# B&R Automation Studio project 8238 (part 18)

#### mnParam_GetCsvDat.st - Parsen einer CSV-Zeile
```iecst
(********************************************************************
 * COPYRIGHT -- Microsoft
 ********************************************************************
 * Library: mnParamLib
 * File: mnParam_GetCsvDat.st
 * Author: hunholz
 * Created: July 25, 2011
 * Changed: Mar 29, 2012
 ********************************************************************
 * Implementation of library mnParamLib
 ********************************************************************)

(* Parsen einer CSV-Zeile *)
FUNCTION_BLOCK mnParam_GetCsvDat

	IF enable THEN

		status := ERR_OK;

		RowType := 0;

		brsmemset(ADR(HeaderVersion), 0, SIZEOF(HeaderVersion));
		brsmemset(ADR(HeaderMachineNo), 0, SIZEOF(HeaderMachineNo));
		brsmemset(ADR(HeaderTime), 0, SIZEOF(HeaderTime));
		brsmemset(ADR(ContainerRow), 0, SIZEOF(ContainerRow));
		brsmemset(ADR(LogicalStructRow), 0, SIZEOF(LogicalStructRow));
		brsmemset(ADR(ParamNumRow), 0, SIZEOF(ParamNumRow));
		brsmemset(ADR(ParamStringRow), 0, SIZEOF(ParamStringRow));
		brsmemset(ADR(CsvNumRow), 0, SIZEOF(CsvNumRow));
		brsmemset(ADR(CsvStringRow), 0, SIZEOF(CsvStringRow));
		brsmemset(ADR(CsvIPRow),0,SIZEOF(CsvIPRow));
		brsmemset(ADR(csvTextRow),0,SIZEOF(csvTextRow));
		brsmemset(ADR(csvHelpTextRow), 0, SIZEOF(csvHelpTextRow));
		brsmemset(ADR(CsvCProw), 0, SIZEOF(CsvCProw));

		_pUtfCsvString := ADR(utfCsvString);

		_GetNextSubstring.enable := TRUE;
		_GetNextSubstring(pUtfCsvString := _pUtfCsvString);

		_utfRowType := "";

		brwcsncpy(ADR(_utfRowType), _GetNextSubstring.pUtfCsvSubstring, MIN(_GetNextSubstring.Length, 15));
		brwcsconv(ADR(_sRowType), ADR(_utfRowType), 1);

		_diRowType := atoi(ADR(_sRowType) );

		IF _diRowType = MNPARAM_CSV_FILEEND THEN

			// FileEnde
			RowType := MNPARAM_CSV_FILEEND;
			// Keine Rückgabewerte

		ELSIF _diRowType = MNPARAM_CSV_COMMENT THEN

			// Kommentarzeile
			RowType := MNPARAM_CSV_COMMENT;

		ELSIF _diRowType = MNPARAM_CSV_HEADER_VERSION THEN

			// Version Datenmodell
			RowType := MNPARAM_CSV_HEADER_VERSION;

			IF NOT _GetNextSubstring.EndOfLine THEN

				_GetNextSubstring(pUtfCsvString := _pUtfCsvString);

				_utfSubString := "";

				brwcsncpy(ADR(_utfSubString), _GetNextSubstring.pUtfCsvSubstring, MIN(_GetNextSubstring.Length, 63));
				brwcsconv(ADR(_sSubString), ADR(_utfSubString), 1);
				_diVersion := atoi(ADR(_sSubString) );

				HeaderVersion.wVersion := DINT_TO_UINT(LIMIT(0, _diVersion, 65535));

			END_IF

			IF NOT _GetNextSubstring.EndOfLine THEN

				_GetNextSubstring(pUtfCsvString := _pUtfCsvString);

				_utfSubString := "";

				brwcsncpy(ADR(_utfSubString), _GetNextSubstring.pUtfCsvSubstring, MIN(_GetNextSubstring.Length, 63));
				brwcsconv(ADR(_sSubString), ADR(_utfSubString), 1);

				_atodt(pStr := ADR(_sSubString));
				HeaderVersion.dtTimestamp := _atodt.dtTimeStamp;

			END_IF

			IF NOT _GetNextSubstring.EndOfLine THEN

				_GetNextSubstring(pUtfCsvString := _pUtfCsvString);

				brwcsncpy(ADR(HeaderVersion.utfMachineType), _GetNextSubstring.pUtfCsvSubstring, MIN(_GetNextSubstring.Length,11));

			END_IF

			IF NOT _GetNextSubstring.EndOfLine THEN

				_GetNextSubstring(pUtfCsvString := _pUtfCsvString);

				brwcsncpy(ADR(HeaderVersion.utfMachineSubType), _GetNextSubstring.pUtfCsvSubstring, MIN(_GetNextSubstring.Length,11));

			END_IF

		ELSIF _diRowType = MNPARAM_CSV_HEADER_MACHINENO THEN

			// Maschinennummer
			RowType := MNPARAM_CSV_HEADER_MACHINENO;

			IF NOT _GetNextSubstring.EndOfLine THEN

				_GetNextSubstring(pUtfCsvString := _pUtfCsvString);

				brwcsncpy(ADR(HeaderMachineNo.utfMachineNo), _GetNextSubstring.pUtfCsvSubstring, MIN(_GetNextSubstring.Length,15));

			END_IF

		ELSIF _diRowType = MNPARAM_CSV_HEADER_TIMESTAMP THEN

			// TimeStamp
			RowType := MNPARAM_CSV_HEADER_TIMESTAMP;

			IF NOT _GetNextSubstring.EndOfLine THEN

				_GetNextSubstring(pUtfCsvString := _pUtfCsvString);

				_utfSubString := "";

				brwcsncpy(ADR(_utfSubString), _GetNextSubstring.pUtfCsvSubstring, MIN(_GetNextSubstring.Length, 63));
				brwcsconv(ADR(_sSubString), ADR(_utfSubString), 1);

				_atodt(pStr := ADR(_sSubString));
				HeaderTime.dtTimestamp := _atodt.dtTimeStamp;

			END_IF

		ELSIF _diRowType = MNPARAM_CSV_LANGUAGEDEF THEN

			// Sprachdefinition
			RowType := MNPARAM_CSV_LANGUAGEDEF;

			IF NOT _GetNextSubstring.EndOfLine THEN

				_GetNextSubstring(pUtfCsvString := _pUtfCsvString);

				_utfSubString := "";

				brwcsncpy(ADR(_utfSubString), _GetNextSubstring.pUtfCsvSubstring, MIN(_GetNextSubstring.Length, 63));
				brwcsconv(ADR(_sSubString), ADR(_utfSubString), 1);
				_diNum := atoi(ADR(_sSubString) );

				CsvLCIDrow.LCID := DINT_TO_UINT(LIMIT(0, _diNum, 65535));

			END_IF

			IF NOT _GetNextSubstring.EndOfLine THEN

				_GetNextSubstring(pUtfCsvString := _pUtfCsvString);

				brwcsncpy(ADR(CsvLCIDrow.utfName), _GetNextSubstring.pUtfCsvSubstring, MIN(_GetNextSubstring.Length, 31));

			END_IF

		ELSIF _diRowType = MNPARAM_CSV_LAN_HELPTEXT THEN

			// Sprachhilfstext
			RowType := MNPARAM_CSV_LAN_HELPTEXT;

			IF NOT _GetNextSubstring.EndOfLine THEN

				_GetNextSubstring(pUtfCsvString := _pUtfCsvString);

				_utfSubString := "";

				brwcsncpy(ADR(_utfSubString), _GetNextSubstring.pUtfCsvSubstring, MIN(_GetNextSubstring.Length, 63));
				brwcsconv(ADR(_sSubString), ADR(_utfSubString), 1);
				_diNum := atoi(ADR(_sSubString) );

				csvHelpTextRow.LCID := DINT_TO_UINT(LIMIT(0, _diNum, 65535));

			END_IF

			IF NOT _GetNextSubstring.EndOfLine THEN

				_GetNextSubstring(pUtfCsvString := _pUtfCsvString);

				_utfSubString := "";

				brwcsncpy(ADR(_utfSubString), _GetNextSubstring.pUtfCsvSubstring, MIN(_GetNextSubstring.Length, 63));
				brwcsconv(ADR(_sSubString), ADR(_utfSubString), 1);
				_diNum := atoi(ADR(_sSubString) );

				csvHelpTextRow.FunctionID := DINT_TO_UINT(LIMIT(0, _diNum, 65535));

			END_IF

			IF NOT _GetNextSubstring.EndOfLine THEN

				_GetNextSubstring(pUtfCsvString := _pUtfCsvString);

				_utfSubString := "";

				brwcsncpy(ADR(_utfSubString), _GetNextSubstring.pUtfCsvSubstring, MIN(_GetNextSubstring.Length, 63));
				brwcsconv(ADR(_sSubString), ADR(_utfSubString), 1);
				_diNum := atoi(ADR(_sSubString) );

				csvHelpTextRow.TextNo := DINT_TO_UINT(LIMIT(0, _diNum, 65535));

			END_IF

			IF NOT _GetNextSubstring.EndOfLine THEN

				_GetNextSubstring(pUtfCsvString := _pUtfCsvString);

				brwcsncpy(ADR(csvHelpTextRow.utfHelpText), _GetNextSubstring.pUtfCsvSubstring, MIN(_GetNextSubstring.Length, 255));

			END_IF

		ELSIF _diRowType = MNPARAM_CSV_LAN_TEXT THEN

			// Sprachtext
			RowType := MNPARAM_CSV_LAN_TEXT;

			IF NOT _GetNextSubstring.EndOfLine THEN

				_GetNextSubstring(pUtfCsvString := _pUtfCsvString);

				_utfSubString := "";

				brwcsncpy(ADR(_utfSubString), _GetNextSubstring.pUtfCsvSubstring, MIN(_GetNextSubstring.Length, 63));
				brwcsconv(ADR(_sSubString), ADR(_utfSubString), 1);
				_diNum := atoi(ADR(_sSubString) );

				csvTextRow.LCID := DINT_TO_UINT(LIMIT(0, _diNum, 65535));

			END_IF

			IF NOT _GetNextSubstring.EndOfLine THEN

				_GetNextSubstring(pUtfCsvString := _pUtfCsvString);

				_utfSubString := "";

				brwcsncpy(ADR(_utfSubString), _GetNextSubstring.pUtfCsvSubstring, MIN(_GetNextSubstring.Length, 63));
				brwcsconv(ADR(_sSubString), ADR(_utfSubString), 1);
				_diNum := atoi(ADR(_sSubString) );

				csvTextRow.FunctionID := DINT_TO_UINT(LIMIT(0, _diNum, 65535));

			END_IF

			IF NOT _GetNextSubstring.EndOfLine THEN

				_GetNextSubstring(pUtfCsvString := _pUtfCsvString);

				_utfSubString := "";

				brwcsncpy(ADR(_utfSubString), _GetNextSubstring.pUtfCsvSubstring, MIN(_GetNextSubstring.Length, 63));
				brwcsconv(ADR(_sSubString), ADR(_utfSubString), 1);
				_diNum := atoi(ADR(_sSubString) );

				csvTextRow.TextNo := DINT_TO_UINT(LIMIT(0, _diNum, 65535));

			END_IF

			IF NOT _GetNextSubstring.EndOfLine THEN

				_GetNextSubstring(pUtfCsvString := _pUtfCsvString);

				brwcsncpy(ADR(csvTextRow.utfText), _GetNextSubstring.pUtfCsvSubstring, MIN(_GetNextSubstring.Length, 63));

			END_IF

		ELSIF _diRowType = MNPARAM_CSV_DEF_CONTAINER THEN

			// Containerbeschreibung
			RowType := MNPARAM_CSV_DEF_CONTAINER;

			// Container ID
			IF NOT _GetNextSubstring.EndOfLine THEN

				_GetNextSubstring(pUtfCsvString := _pUtfCsvString);

				_utfSubString := "";

				brwcsncpy(ADR(_utfSubString), _GetNextSubstring.pUtfCsvSubstring, MIN(_GetNextSubstring.Length, 63));
				brwcsconv(ADR(_sSubString), ADR(_utfSubString), 1);
				_diNum := atoi(ADR(_sSubString) );

				ContainerRow.siContainerID := DINT_TO_SINT(LIMIT(-128, _diNum, 127));

			END_IF

			// DirectParam
			IF NOT _GetNextSubstring.EndOfLine THEN

				_GetNextSubstring(pUtfCsvString := _pUtfCsvString);

				_utfSubString := "";

				brwcsncpy(ADR(_utfSubString), _GetNextSubstring.pUtfCsvSubstring, MIN(_GetNextSubstring.Length, 63));
				brwcsconv(ADR(_sSubString), ADR(_utfSubString), 1);
				_diNum := atoi(ADR(_sSubString) );

				ContainerRow.bDirectParam := DINT_TO_BOOL(LIMIT(0, _diNum, 1));

			END_IF

			// Name Data Obj
			IF NOT _GetNextSubstring.EndOfLine THEN

				_GetNextSubstring(pUtfCsvString := _pUtfCsvString);

				_utfSubString := "";

				brwcsncpy(ADR(_utfDataObj), _GetNextSubstring.pUtfCsvSubstring, MIN(_GetNextSubstring.Length, 11));
				brwcsconv(ADR(ContainerRow.sNameDataObj), ADR(_utfDataObj), 1);

			END_IF

			// Name Csv File
			IF NOT _GetNextSubstring.EndOfLine THEN

				_GetNextSubstring(pUtfCsvString := _pUtfCsvString);

				_utfSubString := "";

				brwcsncpy(ADR(_utfSubString), _GetNextSubstring.pUtfCsvSubstring, MIN(_GetNextSubstring.Length, 31));
				brwcsconv(ADR(ContainerRow.sNameCsv), ADR(_utfSubString), 1);

			END_IF

			// Min Bound
			IF NOT _GetNextSubstring.EndOfLine THEN

				_GetNextSubstring(pUtfCsvString := _pUtfCsvString);

				_utfSubString := "";

				brwcsncpy(ADR(_utfSubString), _GetNextSubstring.pUtfCsvSubstring, MIN(_GetNextSubstring.Length, 63));
				brwcsconv(ADR(_sSubString), ADR(_utfSubString), 1);
				_diNum := atoi(ADR(_sSubString) );

				ContainerRow.wMinBound := DINT_TO_UINT(LIMIT(0, _diNum, 65535));

			END_IF

			// Dimension
			IF NOT _GetNextSubstring.EndOfLine THEN

				_GetNextSubstring(pUtfCsvString := _pUtfCsvString);

				_utfSubString := "";

				brwcsncpy(ADR(_utfSubString), _GetNextSubstring.pUtfCsvSubstring, MIN(_GetNextSubstring.Length, 63));
				brwcsconv(ADR(_sSubString), ADR(_utfSubString), 1);
				_diNum := atoi(ADR(_sSubString) );

				ContainerRow.wDimension := DINT_TO_UINT(LIMIT(0, _diNum, 65535));

			END_IF

			// Struct Root
			IF NOT _GetNextSubstring.EndOfLine THEN

				_GetNextSubstring(pUtfCsvString := _pUtfCsvString);

				_utfSubString := "";

				brwcsncpy(ADR(_utfSubString), _GetNextSubstring.pUtfCsvSubstring, MIN(_GetNextSubstring.Length, 31));
				brwcsconv(ADR(ContainerRow.sStrucRoot), ADR(_utfSubString), 1);

			END_IF

			IF NOT _GetNextSubstring.EndOfLine THEN
				_GetNextSubstring(pUtfCsvString := _pUtfCsvString);
			END_IF

			// Anzahl der Numparameter
			IF NOT _GetNextSubstring.EndOfLine THEN

				_GetNextSubstring(pUtfCsvString := _pUtfCsvString);

				_utfSubString := "";

				brwcsncpy(ADR(_utfSubString), _GetNextSubstring.pUtfCsvSubstring, MIN(_GetNextSubstring.Length, 63));
				brwcsconv(ADR(_sSubString), ADR(_utfSubString), 1);

				ContainerRow.lCountNum := atoi(ADR(_sSubString) );

			END_IF

			// Anzahl der Stringparameter
			IF NOT _GetNextSubstring.EndOfLine THEN

				_GetNextSubstring(pUtfCsvString := _pUtfCsvString);

				_utfSubString := "";

				brwcsncpy(ADR(_utfSubString), _GetNextSubstring.pUtfCsvSubstring, MIN(_GetNextSubstring.Length, 63));
				brwcsconv(ADR(_sSubString), ADR(_utfSubString), 1);

				ContainerRow.lCountString := atoi(ADR(_sSubString) );

			END_IF

		ELSIF _diRowType = MNPARAM_CSV_DEF_LOGSTRUC THEN

			// Logische Struktur
			RowType := MNPARAM_CSV_DEF_LOGSTRUC;

			// Index
			IF NOT _GetNextSubstring.EndOfLine THEN

				_GetNextSubstring(pUtfCsvString := _pUtfCsvString);

				_utfSubString := "";

				brwcsncpy(ADR(_utfSubString), _GetNextSubstring.pUtfCsvSubstring, MIN(_GetNextSubstring.Length, 63));
				brwcsconv(ADR(_sSubString), ADR(_utfSubString), 1);
				_diNum := atoi(ADR(_sSubString) );

				LogicalStructRow.wLogStrucNo := DINT_TO_UINT(LIMIT(0, _diNum, 65535));

			END_IF

			// Min Bound
			IF NOT _GetNextSubstring.EndOfLine THEN

				_GetNextSubstring(pUtfCsvString := _pUtfCsvString);

				_utfSubString := "";

				brwcsncpy(ADR(_utfSubString), _GetNextSubstring.pUtfCsvSubstring, MIN(_GetNextSubstring.Length, 63));
				brwcsconv(ADR(_sSubString), ADR(_utfSubString), 1);
				_diNum := atoi(ADR(_sSubString) );

				LogicalStructRow.wMinBound := DINT_TO_UINT(LIMIT(0, _diNum, 65535));

			END_IF

			// Dimension
			IF NOT _GetNextSubstring.EndOfLine THEN

				_GetNextSubstring(pUtfCsvString := _pUtfCsvString);

				_utfSubString := "";

				brwcsncpy(ADR(_utfSubString), _GetNextSubstring.pUtfCsvSubstring, MIN(_GetNextSubstring.Length, 63));
				brwcsconv(ADR(_sSubString), ADR(_utfSubString), 1);
				_diNum := atoi(ADR(_sSubString) );

				LogicalStructRow.wDimension := DINT_TO_UINT(LIMIT(0, _diNum, 65535));

			END_IF

			// Referenz
			IF NOT _GetNextSubstring.EndOfLine THEN

				_GetNextSubstring(pUtfCsvString := _pUtfCsvString);

				_utfSubString := "";

				brwcsncpy(ADR(_utfSubString), _GetNextSubstring.pUtfCsvSubstring, MIN(_GetNextSubstring.Length, 63));
				brwcsconv(ADR(_sSubString), ADR(_utfSubString), 1);
				_diNum := atoi(ADR(_sSubString) );

				LogicalStructRow.iReferenz := DINT_TO_INT(LIMIT(-32768, _diNum, 32767));

			END_IF

			// Ref Visible
			IF NOT _GetNextSubstring.EndOfLine THEN

				_GetNextSubstring(pUtfCsvString := _pUtfCsvString);

				_utfSubString := "";

				brwcsncpy(ADR(_utfSubString), _GetNextSubstring.pUtfCsvSubstring, MIN(_GetNextSubstring.Length, 63));
				brwcsconv(ADR(_sSubString), ADR(_utfSubString), 1);
				_diNum := atoi(ADR(_sSubString) );

				LogicalStructRow.wRefVisible := DINT_TO_UINT(LIMIT(0, _diNum, 65535));

			END_IF

			// Ref Text
			IF NOT _GetNextSubstring.EndOfLine THEN

				_GetNextSubstring(pUtfCsvString := _pUtfCsvString);

				_utfSubString := "";

				brwcsncpy(ADR(_utfSubString), _GetNextSubstring.pUtfCsvSubstring, MIN(_GetNextSubstring.Length, 63));
				brwcsconv(ADR(_sSubString), ADR(_utfSubString), 1);
				_diNum := atoi(ADR(_sSubString) );

				LogicalStructRow.wRefText := DINT_TO_UINT(LIMIT(0, _diNum, 65535));

			END_IF

			// WriteAccess
			IF NOT _GetNextSubstring.EndOfLine THEN

				_GetNextSubstring(pUtfCsvString := _pUtfCsvString);

				_utfSubString := "";

				brwcsncpy(ADR(_utfSubString), _GetNextSubstring.pUtfCsvSubstring, MIN(_GetNextSubstring.Length, 63));
				brwcsconv(ADR(_sSubString), ADR(_utfSubString), 1);
				_diNum := atoi(ADR(_sSubString) );

				LogicalStructRow.siWriteAccess := DINT_TO_SINT(LIMIT(-128, _diNum, 127));

			END_IF

			// VisibleAccess
			IF NOT _GetNextSubstring.EndOfLine THEN

				_GetNextSubstring(pUtfCsvString := _pUtfCsvString);

				_utfSubString := "";

				brwcsncpy(ADR(_utfSubString), _GetNextSubstring.pUtfCsvSubstring, MIN(_GetNextSubstring.Length, 63));
				brwcsconv(ADR(_sSubString), ADR(_utfSubString), 1);
				_diNum := atoi(ADR(_sSubString) );

				LogicalStructRow.siVisibleAccess := DINT_TO_SINT(LIMIT(-128, _diNum, 127));

			END_IF

			// Format Array
			IF NOT _GetNextSubstring.EndOfLine THEN

				_GetNextSubstring(pUtfCsvString := _pUtfCsvString);

				_utfSubString := "";

				brwcsncpy(ADR(_utfSubString), _GetNextSubstring.pUtfCsvSubstring, MIN(_GetNextSubstring.Length, 63));
				brwcsconv(ADR(_sSubString), ADR(_utfSubString), 1);
				_diNum := atoi(ADR(_sSubString) );

				LogicalStructRow.bFormatArray := DINT_TO_USINT(LIMIT(0, _diNum, 255));

			END_IF

			// Machine Sub Type
			IF NOT _GetNextSubstring.EndOfLine THEN

				_GetNextSubstring(pUtfCsvString := _pUtfCsvString);

				brwcsncpy(ADR(LogicalStructRow.utfMachineSubType), _GetNextSubstring.pUtfCsvSubstring, MIN(_GetNextSubstring.Length, 11));

			END_IF

			// LogStructName
			IF NOT _GetNextSubstring.EndOfLine THEN

				_GetNextSubstring(pUtfCsvString := _pUtfCsvString);

				brwcsncpy(ADR(LogicalStructRow.utfLogStrucName), _GetNextSubstring.pUtfCsvSubstring, MIN(_GetNextSubstring.Length, 31));

			END_IF

		ELSIF _diRowType = MNPARAM_CSV_DEF_STRING THEN

			// String
			RowType := MNPARAM_CSV_DEF_STRING;

			// Index
			IF NOT _GetNextSubstring.EndOfLine THEN

				_GetNextSubstring(pUtfCsvString := _pUtfCsvString);

				_utfSubString := "";

				brwcsncpy(ADR(_utfSubString), _GetNextSubstring.pUtfCsvSubstring, MIN(_GetNextSubstring.Length, 63));
				brwcsconv(ADR(_sSubString), ADR(_utfSubString), 1);
				_diNum := atoi(ADR(_sSubString) );

				ParamStringRow.wIdxStringPar := DINT_TO_UINT(LIMIT(0, _diNum, 65535));

			END_IF

			// Function ID
			IF NOT _GetNextSubstring.EndOfLine THEN

				_GetNextSubstring(pUtfCsvString := _pUtfCsvString);

				_utfSubString := "";

				brwcsncpy(ADR(_utfSubString), _GetNextSubstring.pUtfCsvSubstring, MIN(_GetNextSubstring.Length, 63));
				brwcsconv(ADR(_sSubString), ADR(_utfSubString), 1);
				_diNum := atoi(ADR(_sSubString) );

				ParamStringRow.wFunction_ID := DINT_TO_UINT(LIMIT(0, _diNum, 65535));

			END_IF

			// Parameter No
			IF NOT _GetNextSubstring.EndOfLine THEN

				_GetNextSubstring(pUtfCsvString := _pUtfCsvString);

				_utfSubString := "";

				brwcsncpy(ADR(_utfSubString), _GetNextSubstring.pUtfCsvSubstring, MIN(_GetNextSubstring.Length, 63));
				brwcsconv(ADR(_sSubString), ADR(_utfSubString), 1);
				_diNum := atoi(ADR(_sSubString) );

				ParamStringRow.wParNo := DINT_TO_UINT(LIMIT(0, _diNum, 65535));

			END_IF

			// Länge
			IF NOT _GetNextSubstring.EndOfLine THEN

				_GetNextSubstring(pUtfCsvString := _pUtfCsvString);

				_utfSubString := "";

				brwcsncpy(ADR(_utfSubString), _GetNextSubstring.pUtfCsvSubstring, MIN(_GetNextSubstring.Length, 63));
				brwcsconv(ADR(_sSubString), ADR(_utfSubString), 1);
				_diNum := atoi(ADR(_sSubString) );

				ParamStringRow.bLenght := DINT_TO_USINT(LIMIT(0, _diNum, 255));

			END_IF

			// WriteAccess
			IF NOT _GetNextSubstring.EndOfLine THEN

				_GetNextSubstring(pUtfCsvString := _pUtfCsvString);

				_utfSubString := "";

				brwcsncpy(ADR(_utfSubString), _GetNextSubstring.pUtfCsvSubstring, MIN(_GetNextSubstring.Length, 63));
				brwcsconv(ADR(_sSubString), ADR(_utfSubString), 1);
				_diNum := atoi(ADR(_sSubString) );

				ParamStringRow.siWriteAccess := DINT_TO_SINT(LIMIT(-128, _diNum, 127));

			END_IF

			// VisibleAccess
			IF NOT _GetNextSubstring.EndOfLine THEN

				_GetNextSubstring(pUtfCsvString := _pUtfCsvString);

				_utfSubString := "";

				brwcsncpy(ADR(_utfSubString), _GetNextSubstring.pUtfCsvSubstring, MIN(_GetNextSubstring.Length, 63));
				brwcsconv(ADR(_sSubString), ADR(_utfSubString), 1);
				_diNum := atoi(ADR(_sSubString) );

				ParamStringRow.siVisibleAccess := DINT_TO_SINT(LIMIT(-128, _diNum, 127));

			END_IF

			// Adresse
			IF NOT _GetNextSubstring.EndOfLine THEN

				_GetNextSubstring(pUtfCsvString := _pUtfCsvString);

				_utfSubString := "";

				brwcsncpy(ADR(_utfSubString), _GetNextSubstring.pUtfCsvSubstring, MIN(_GetNextSubstring.Length, 63));
				brwcsconv(ADR(ParamStringRow.sAdresse), ADR(_utfSubString), 1);

			END_IF

			// Min Bound
			IF NOT _GetNextSubstring.EndOfLine THEN

				_GetNextSubstring(pUtfCsvString := _pUtfCsvString);

				_utfSubString := "";

				brwcsncpy(ADR(_utfSubString), _GetNextSubstring.pUtfCsvSubstring, MIN(_GetNextSubstring.Length, 63));
				brwcsconv(ADR(_sSubString), ADR(_utfSubString), 1);
				_diNum := atoi(ADR(_sSubString) );

				ParamStringRow.wMinBound := DINT_TO_UINT(LIMIT(0, _diNum, 65535));

			END_IF

			// Dimension
			IF NOT _GetNextSubstring.EndOfLine THEN

				_GetNextSubstring(pUtfCsvString := _pUtfCsvString);

				_utfSubString := "";

				brwcsncpy(ADR(_utfSubString), _GetNextSubstring.pUtfCsvSubstring, MIN(_GetNextSubstring.Length, 63));
				brwcsconv(ADR(_sSubString), ADR(_utfSubString), 1);
				_diNum := atoi(ADR(_sSubString) );

				ParamStringRow.wDimension := DINT_TO_UINT(LIMIT(0, _diNum, 65535));

			END_IF

			// Referenz
			IF NOT _GetNextSubstring.EndOfLine THEN

				_GetNextSubstring(pUtfCsvString := _pUtfCsvString);

				_utfSubString := "";

				brwcsncpy(ADR(_utfSubString), _GetNextSubstring.pUtfCsvSubstring, MIN(_GetNextSubstring.Length, 63));
				brwcsconv(ADR(_sSubString), ADR(_utfSubString), 1);
				_diNum := atoi(ADR(_sSubString) );

				ParamStringRow.wReferenz := DINT_TO_UINT(LIMIT(0, _diNum, 65535));

			END_IF

			// Def. Value
			IF NOT _GetNextSubstring.EndOfLine THEN

				_GetNextSubstring(pUtfCsvString := _pUtfCsvString);

				brwcsncpy(ADR(ParamStringRow.utfDefValue), _GetNextSubstring.pUtfCsvSubstring, MIN(_GetNextSubstring.Length, 31));

			END_IF

			// Machine Sub Type
			IF NOT _GetNextSubstring.EndOfLine THEN

				_GetNextSubstring(pUtfCsvString := _pUtfCsvString);

				brwcsncpy(ADR(ParamStringRow.utfMachineSubType), _GetNextSubstring.pUtfCsvSubstring, MIN(_GetNextSubstring.Length, 11));

			END_IF

			// RefVisible
			IF NOT _GetNextSubstring.EndOfLine THEN

				_GetNextSubstring(pUtfCsvString := _pUtfCsvString);

				_utfSubString := "";

				brwcsncpy(ADR(_utfSubString), _GetNextSubstring.pUtfCsvSubstring, MIN(_GetNextSubstring.Length, 63));
				brwcsconv(ADR(_sSubString), ADR(_utfSubString), 1);
				_diNum := atoi(ADR(_sSubString) );

				ParamStringRow.wRefVisible := DINT_TO_UINT(LIMIT(0, _diNum, 65535));

			END_IF

			// RefVisible
			IF NOT _GetNextSubstring.EndOfLine THEN

				_GetNextSubstring(pUtfCsvString := _pUtfCsvString);

				_utfSubString := "";

				brwcsncpy(ADR(_utfSubString), _GetNextSubstring.pUtfCsvSubstring, MIN(_GetNextSubstring.Length, 63));
				brwcsconv(ADR(_sSubString), ADR(_utfSubString), 1);
				_diNum := atoi(ADR(_sSubString) );

				ParamStringRow.wRefVisibleType := DINT_TO_UINT(LIMIT(0, _diNum, 65535));

			END_IF

			// RefText
			IF NOT _GetNextSubstring.EndOfLine THEN

				_GetNextSubstring(pUtfCsvString := _pUtfCsvString);

				_utfSubString := "";

				brwcsncpy(ADR(_utfSubString), _GetNextSubstring.pUtfCsvSubstring, MIN(_GetNextSubstring.Length, 63));
				brwcsconv(ADR(_sSubString), ADR(_utfSubString), 1);
				_diNum := atoi(ADR(_sSubString) );

				ParamStringRow.wRefText := DINT_TO_UINT(LIMIT(0, _diNum, 65535));

			END_IF

		ELSIF _diRowType = MNPARAM_CSV_DEF_NUM OR _diRowType = MNPARAM_CSV_DEF_REAL THEN

			// Logische Struktur
			RowType := DINT_TO_UINT(_diRowType);
			ParamNumRow.bRowType := UINT_TO_USINT(RowType - MNPARAM_CSV_DEF_NUM);

			// Index
			IF NOT _GetNextSubstring.EndOfLine THEN

				_GetNextSubstring(pUtfCsvString := _pUtfCsvString);

				_utfSubString := "";

				brwcsncpy(ADR(_utfSubString), _GetNextSubstring.pUtfCsvSubstring, MIN(_GetNextSubstring.Length, 63));
				brwcsconv(ADR(_sSubString), ADR(_utfSubString), 1);
				_diNum := atoi(ADR(_sSubString) );

				ParamNumRow.wIdxNumPar := DINT_TO_UINT(LIMIT(0, _diNum, 65535));

			END_IF

			// Function ID
			IF NOT _GetNextSubstring.EndOfLine THEN

				_GetNextSubstring(pUtfCsvString := _pUtfCsvString);

				_utfSubString := "";

				brwcsncpy(ADR(_utfSubString), _GetNextSubstring.pUtfCsvSubstring, MIN(_GetNextSubstring.Length, 63));
				brwcsconv(ADR(_sSubString), ADR(_utfSubString), 1);
				_diNum := atoi(ADR(_sSubString) );

				ParamNumRow.wFunction_ID := DINT_TO_UINT(LIMIT(0, _diNum, 65535));

			END_IF

			// Parameter No
			IF NOT _GetNextSubstring.EndOfLine THEN

				_GetNextSubstring(pUtfCsvString := _pUtfCsvString);

				_utfSubString := "";

				brwcsncpy(ADR(_utfSubString), _GetNextSubstring.pUtfCsvSubstring, MIN(_GetNextSubstring.Length, 63));
				brwcsconv(ADR(_sSubString), ADR(_utfSubString), 1);
				_diNum := atoi(ADR(_sSubString) );

				ParamNumRow.wParNo := DINT_TO_UINT(LIMIT(0, _diNum, 65535));

			END_IF

			// WriteAccess
			IF NOT _GetNextSubstring.EndOfLine THEN

				_GetNextSubstring(pUtfCsvString := _pUtfCsvString);

				_utfSubString := "";

				brwcsncpy(ADR(_utfSubString), _GetNextSubstring.pUtfCsvSubstring, MIN(_GetNextSubstring.Length, 63));
				brwcsconv(ADR(_sSubString), ADR(_utfSubString), 1);
				_diNum := atoi(ADR(_sSubString) );

				ParamNumRow.siWriteAccess := DINT_TO_SINT(LIMIT(-128, _diNum, 127));

			END_IF

			// VisibleAccess
			IF NOT _GetNextSubstring.EndOfLine THEN

				_GetNextSubstring(pUtfCsvString := _pUtfCsvString);

				_utfSubString := "";

				brwcsncpy(ADR(_utfSubString), _GetNextSubstring.pUtfCsvSubstring, MIN(_GetNextSubstring.Length, 63));
				brwcsconv(ADR(_sSubString), ADR(_utfSubString), 1);
				_diNum := atoi(ADR(_sSubString) );

				ParamNumRow.siVisibleAccess := DINT_TO_SINT(LIMIT(-128, _diNum, 127));

			END_IF

			// Unit ID
			IF NOT _GetNextSubstring.EndOfLine THEN

				_GetNextSubstring(pUtfCsvString := _pUtfCsvString);

				_utfSubString := "";

				brwcsncpy(ADR(_utfSubString), _GetNextSubstring.pUtfCsvSubstring, MIN(_GetNextSubstring.Length, 63));
				brwcsconv(ADR(_sSubString), ADR(_utfSubString), 1);
				_diNum := atoi(ADR(_sSubString) );

				ParamNumRow.wUnitID := DINT_TO_UINT(LIMIT(0, _diNum, 65535));

			END_IF

			// Adresse
			IF NOT _GetNextSubstring.EndOfLine THEN

				_GetNextSubstring(pUtfCsvString := _pUtfCsvString);

				_utfSubString := "";

				brwcsncpy(ADR(_utfSubString), _GetNextSubstring.pUtfCsvSubstring, MIN(_GetNextSubstring.Length, 63));
				brwcsconv(ADR(ParamNumRow.sAdresse), ADR(_utfSubString), 1);

			END_IF

			// Min Bound
			IF NOT _GetNextSubstring.EndOfLine THEN

				_GetNextSubstring(pUtfCsvString := _pUtfCsvString);

				_utfSubString := "";

				brwcsncpy(ADR(_utfSubString), _GetNextSubstring.pUtfCsvSubstring, MIN(_GetNextSubstring.Length, 63));
				brwcsconv(ADR(_sSubString), ADR(_utfSubString), 1);
				_diNum := atoi(ADR(_sSubString) );

				ParamNumRow.wMinBound := DINT_TO_UINT(LIMIT(0, _diNum, 65535));

			END_IF

			// Dimension
			IF NOT _GetNextSubstring.EndOfLine THEN

				_GetNextSubstring(pUtfCsvString := _pUtfCsvString);

				_utfSubString := "";

				brwcsncpy(ADR(_utfSubString), _GetNextSubstring.pUtfCsvSubstring, MIN(_GetNextSubstring.Length, 63));
				brwcsconv(ADR(_sSubString), ADR(_utfSubString), 1);
				_diNum := atoi(ADR(_sSubString) );

				ParamNumRow.wDimension := DINT_TO_UINT(LIMIT(0, _diNum, 65535));

			END_IF

			// Referenz
			IF NOT _GetNextSubstring.EndOfLine THEN

				_GetNextSubstring(pUtfCsvString := _pUtfCsvString);

				_utfSubString := "";

				brwcsncpy(ADR(_utfSubString), _GetNextSubstring.pUtfCsvSubstring, MIN(_GetNextSubstring.Length, 63));
				brwcsconv(ADR(_sSubString), ADR(_utfSubString), 1);
				_diNum := atoi(ADR(_sSubString) );

				ParamNumRow.wReferenz := DINT_TO_UINT(LIMIT(0, _diNum, 65535));

			END_IF

			IF ParamNumRow.bRowType = 0 THEN

				// MinValue
				IF NOT _GetNextSubstring.EndOfLine THEN

					_GetNextSubstring(pUtfCsvString := _pUtfCsvString);

					_utfSubString := "";

					brwcsncpy(ADR(_utfSubString), _GetNextSubstring.pUtfCsvSubstring, MIN(_GetNextSubstring.Length, 63));
					brwcsconv(ADR(_sSubString), ADR(_utfSubString), 1);
					ParamNumRow.diMinValue := atoi(ADR(_sSubString) );

				END_IF

				// MaxValue
				IF NOT _GetNextSubstring.EndOfLine THEN

					_GetNextSubstring(pUtfCsvString := _pUtfCsvString);

					_utfSubString := "";

					brwcsncpy(ADR(_utfSubString), _GetNextSubstring.pUtfCsvSubstring, MIN(_GetNextSubstring.Length, 63));
					brwcsconv(ADR(_sSubString), ADR(_utfSubString), 1);
					ParamNumRow.diMaxValue := atoi(ADR(_sSubString) );

				END_IF

				// DefValue
				IF NOT _GetNextSubstring.EndOfLine THEN

					_GetNextSubstring(pUtfCsvString := _pUtfCsvString);

					_utfSubString := "";

					brwcsncpy(ADR(_utfSubString), _GetNextSubstring.pUtfCsvSubstring, MIN(_GetNextSubstring.Length, 63));
					brwcsconv(ADR(_sSubString), ADR(_utfSubString), 1);
					ParamNumRow.diDefValue := brsatoi(ADR(_sSubString) );

				END_IF

			ELSE

				// MinValue
				IF NOT _GetNextSubstring.EndOfLine THEN

					_GetNextSubstring(pUtfCsvString := _pUtfCsvString);

					_utfSubString := "";

					brwcsncpy(ADR(_utfSubString), _GetNextSubstring.pUtfCsvSubstring, MIN(_GetNextSubstring.Length, 63));
					brwcsconv(ADR(_sSubString), ADR(_utfSubString), 1);
					_rValue := brsatof(ADR(_sSubString) );
					_pdiValue ACCESS ADR(_rValue);
					ParamNumRow.diMinValue := _pdiValue;

				END_IF

				// MaxValue
				IF NOT _GetNextSubstring.EndOfLine THEN

					_GetNextSubstring(pUtfCsvString := _pUtfCsvString);

					_utfSubString := "";

					brwcsncpy(ADR(_utfSubString), _GetNextSubstring.pUtfCsvSubstring, MIN(_GetNextSubstring.Length, 63));
					brwcsconv(ADR(_sSubString), ADR(_utfSubString), 1);
					_rValue := brsatof(ADR(_sSubString) );
					_pdiValue ACCESS ADR(_rValue);
					ParamNumRow.diMaxValue := _pdiValue;

				END_IF

				// DefValue
				IF NOT _GetNextSubstring.EndOfLine THEN

					_GetNextSubstring(pUtfCsvString := _pUtfCsvString);

					_utfSubString := "";

					brwcsncpy(ADR(_utfSubString), _GetNextSubstring.pUtfCsvSubstring, MIN(_GetNextSubstring.Length, 63));
					brwcsconv(ADR(_sSubString), ADR(_utfSubString), 1);
					_rValue := brsatof(ADR(_sSubString) );
					_pdiValue ACCESS ADR(_rValue);
					ParamNumRow.diDefValue := _pdiValue;

				END_IF

			END_IF

			// InputType
			IF NOT _GetNextSubstring.EndOfLine THEN

				_GetNextSubstring(pUtfCsvString := _pUtfCsvString);

				_utfSubString := "";

				brwcsncpy(ADR(_utfSubString), _GetNextSubstring.pUtfCsvSubstring, MIN(_GetNextSubstring.Length, 63));
				brwcsconv(ADR(_sSubString), ADR(_utfSubString), 1);
				_diNum := atoi(ADR(_sSubString) );

				ParamNumRow.bInputType := DINT_TO_USINT(LIMIT(0, _diNum, 255));

			END_IF

			// ITidx
			IF NOT _GetNextSubstring.EndOfLine THEN

				_GetNextSubstring(pUtfCsvString := _pUtfCsvString);

				_utfSubString := "";

				brwcsncpy(ADR(_utfSubString), _GetNextSubstring.pUtfCsvSubstring, MIN(_GetNextSubstring.Length, 63));
				brwcsconv(ADR(_sSubString), ADR(_utfSubString), 1);
				_diNum := atoi(ADR(_sSubString) );

				ParamNumRow.wITIdx := DINT_TO_UINT(LIMIT(0, _diNum, 65535));

			END_IF

			// Machine Sub Type
			IF NOT _GetNextSubstring.EndOfLine THEN

				_GetNextSubstring(pUtfCsvString := _pUtfCsvString);

				brwcsncpy(ADR(ParamNumRow.utfMachineSubType), _GetNextSubstring.pUtfCsvSubstring, MIN(_GetNextSubstring.Length, 11));

			END_IF

			// RefVisible
			IF NOT _GetNextSubstring.EndOfLine THEN

				_GetNextSubstring(pUtfCsvString := _pUtfCsvString);

				_utfSubString := "";

				brwcsncpy(ADR(_utfSubString), _GetNextSubstring.pUtfCsvSubstring, MIN(_GetNextSubstring.Length, 63));
				brwcsconv(ADR(_sSubString), ADR(_utfSubString), 1);
				_diNum := atoi(ADR(_sSubString) );

				ParamNumRow.wRefVisible := DINT_TO_UINT(LIMIT(0, _diNum, 65535));

			END_IF

			// RefVisibleType
			IF NOT _GetNextSubstring.EndOfLine THEN

				_GetNextSubstring(pUtfCsvString := _pUtfCsvString);

				_utfSubString := "";

				brwcsncpy(ADR(_utfSubString), _GetNextSubstring.pUtfCsvSubstring, MIN(_GetNextSubstring.Length, 63));
				brwcsconv(ADR(_sSubString), ADR(_utfSubString), 1);
				_diNum := atoi(ADR(_sSubString) );

				ParamNumRow.wRefVisibleType := DINT_TO_UINT(LIMIT(0, _diNum, 65535));

			END_IF

			// RefText
			IF NOT _GetNextSubstring.EndOfLine THEN

				_GetNextSubstring(pUtfCsvString := _pUtfCsvString);

				_utfSubString := "";

				brwcsncpy(ADR(_utfSubString), _GetNextSubstring.pUtfCsvSubstring, MIN(_GetNextSubstring.Length, 63));
				brwcsconv(ADR(_sSubString), ADR(_utfSubString), 1);
				_diNum := atoi(ADR(_sSubString) );

				ParamNumRow.wRefText := DINT_TO_UINT(LIMIT(0, _diNum, 65535));

			END_IF

		ELSIF _diRowType = MNPARAM_CSV_IP THEN

			// CSV IP Row
			RowType := MNPARAM_CSV_IP;

			IF NOT _GetNextSubstring.EndOfLine THEN

				_GetNextSubstring(pUtfCsvString := _pUtfCsvString);

				brwcsncpy(ADR(CsvIPRow.utfIP_Adress), _GetNextSubstring.pUtfCsvSubstring, MIN(_GetNextSubstring.Length, 15));

			END_IF

			IF NOT _GetNextSubstring.EndOfLine THEN

				_GetNextSubstring(pUtfCsvString := _pUtfCsvString);

				brwcsncpy(ADR(CsvIPRow.utfGateway), _GetNextSubstring.pUtfCsvSubstring, MIN(_GetNextSubstring.Length, 15));

			END_IF

		ELSIF _diRowType = MNPARAM_CSV_CP THEN

			// CSV Category-Program-Row
			RowType := MNPARAM_CSV_CP;

			// Categroy
			IF NOT _GetNextSubstring.EndOfLine THEN

				_GetNextSubstring(pUtfCsvString := _pUtfCsvString);

				_utfSubString := "";
				brwcsncpy(ADR(_utfSubString), _GetNextSubstring.pUtfCsvSubstring, MIN(_GetNextSubstring.Length, 11));
				CsvCProw.sCategory := WSTRING_TO_STRING(_utfSubString);

			END_IF

			// Category-Name
			IF NOT _GetNextSubstring.EndOfLine THEN

				_GetNextSubstring(pUtfCsvString := _pUtfCsvString);

				brwcsncpy(ADR(CsvCProw.utfCategoryName), _GetNextSubstring.pUtfCsvSubstring, MIN(_GetNextSubstring.Length, 31));

			END_IF

			// Programmno
			IF NOT _GetNextSubstring.EndOfLine THEN

				_GetNextSubstring(pUtfCsvString := _pUtfCsvString);

				_utfSubString := "";

				brwcsncpy(ADR(_utfSubString), _GetNextSubstring.pUtfCsvSubstring, MIN(_GetNextSubstring.Length, 63));
				brwcsconv(ADR(_sSubString), ADR(_utfSubString), 1);
				_diNum := atoi(ADR(_sSubString) );

				CsvCProw.wProgramNo := DINT_TO_UINT(LIMIT(0, _diNum, 65535));

			END_IF

			// Zeitstempel
			IF NOT _GetNextSubstring.EndOfLine THEN

				_GetNextSubstring(pUtfCsvString := _pUtfCsvString);

				_utfSubString := "";

				brwcsncpy(ADR(_utfSubString), _GetNextSubstring.pUtfCsvSubstring, MIN(_GetNextSubstring.Length, 63));
				brwcsconv(ADR(_sSubString), ADR(_utfSubString), 1);

				_atodt(pStr := ADR(_sSubString));
				CsvCProw.dtTimeStamp := _atodt.dtTimeStamp;

			END_IF

			// Verschmutzungsfaktor
			IF NOT _GetNextSubstring.EndOfLine THEN

				_GetNextSubstring(pUtfCsvString := _pUtfCsvString);

				_utfSubString := "";

				brwcsncpy(ADR(_utfSubString), _GetNextSubstring.pUtfCsvSubstring, MIN(_GetNextSubstring.Length, 63));
				brwcsconv(ADR(_sSubString), ADR(_utfSubString), 1);

				CsvCProw.rSoilfactor := STRING_TO_REAL(_sSubString);

			END_IF

			// Beladegrad
			IF NOT _GetNextSubstring.EndOfLine THEN

				_GetNextSubstring(pUtfCsvString := _pUtfCsvString);

				_utfSubString := "";

				brwcsncpy(ADR(_utfSubString), _GetNextSubstring.pUtfCsvSubstring, MIN(_GetNextSubstring.Length, 63));
				brwcsconv(ADR(_sSubString), ADR(_utfSubString), 1);

				CsvCProw.wLoadrate := STRING_TO_UINT(_sSubString);

			END_IF

			// Fordergrundfarbe
			IF NOT _GetNextSubstring.EndOfLine THEN

				_GetNextSubstring(pUtfCsvString := _pUtfCsvString);

				_utfSubString := "";

				brwcsncpy(ADR(_utfSubString), _GetNextSubstring.pUtfCsvSubstring, MIN(_GetNextSubstring.Length, 63));
				brwcsconv(ADR(_sSubString), ADR(_utfSubString), 1);

				CsvCProw.wColFor := STRING_TO_UINT(_sSubString);

			END_IF

			// Hintergrundfarbe
			IF NOT _GetNextSubstring.EndOfLine THEN

				_GetNextSubstring(pUtfCsvString := _pUtfCsvString);

				_utfSubString := "";

				brwcsncpy(ADR(_utfSubString), _GetNextSubstring.pUtfCsvSubstring, MIN(_GetNextSubstring.Length, 63));
				brwcsconv(ADR(_sSubString), ADR(_utfSubString), 1);

				CsvCProw.wColBack := STRING_TO_UINT(_sSubString);

			END_IF

		ELSIF _diRowType = MNPARAM_CSV_DAT_STRING THEN

			// CSV String Parameter
			RowType := MNPARAM_CSV_DAT_STRING;

			// Index
			IF NOT _GetNextSubstring.EndOfLine THEN

				_GetNextSubstring(pUtfCsvString := _pUtfCsvString);

				_utfSubString := "";

				brwcsncpy(ADR(_utfSubString), _GetNextSubstring.pUtfCsvSubstring, MIN(_GetNextSubstring.Length, 63));
				brwcsconv(ADR(_sSubString), ADR(_utfSubString), 1);
				_diNum := atoi(ADR(_sSubString) );

				CsvStringRow.wIdxStringPar := DINT_TO_UINT(LIMIT(0, _diNum, 65535));

			END_IF

			// Value
			IF NOT _GetNextSubstring.EndOfLine THEN

				_GetNextSubstring(pUtfCsvString := _pUtfCsvString);

				brwcsncpy(ADR(CsvStringRow.utfValue), _GetNextSubstring.pUtfCsvSubstring, MIN(_GetNextSubstring.Length, 31));

			END_IF

			//  ArrIndex1
			IF NOT _GetNextSubstring.EndOfLine THEN

				_GetNextSubstring(pUtfCsvString := _pUtfCsvString);

				_utfSubString := "";

				brwcsncpy(ADR(_utfSubString), _GetNextSubstring.pUtfCsvSubstring, MIN(_GetNextSubstring.Length, 63));
				brwcsconv(ADR(_sSubString), ADR(_utfSubString), 1);
				_diNum := atoi(ADR(_sSubString) );

				CsvStringRow.wArrIdx1 := DINT_TO_UINT(LIMIT(0, _diNum, 65535));

			END_IF

			//  ArrIndex2
			IF NOT _GetNextSubstring.EndOfLine THEN

				_GetNextSubstring(pUtfCsvString := _pUtfCsvString);

				_utfSubString := "";

				brwcsncpy(ADR(_utfSubString), _GetNextSubstring.pUtfCsvSubstring, MIN(_GetNextSubstring.Length, 63));
				brwcsconv(ADR(_sSubString), ADR(_utfSubString), 1);
				_diNum := atoi(ADR(_sSubString) );

				CsvStringRow.wArrIdx2 := DINT_TO_UINT(LIMIT(0, _diNum, 65535));

			END_IF

			//  ArrIndex3
			IF NOT _GetNextSubstring.EndOfLine THEN

				_GetNextSubstring(pUtfCsvString := _pUtfCsvString);

				_utfSubString := "";

				brwcsncpy(ADR(_utfSubString), _GetNextSubstring.pUtfCsvSubstring, MIN(_GetNextSubstring.Length, 63));
				brwcsconv(ADR(_sSubString), ADR(_utfSubString), 1);
				_diNum := atoi(ADR(_sSubString) );

				CsvStringRow.wArrIdx3 := DINT_TO_UINT(LIMIT(0, _diNum, 65535));

			END_IF

			//  ArrIndex4
			IF NOT _GetNextSubstring.EndOfLine THEN

				_GetNextSubstring(pUtfCsvString := _pUtfCsvString);

				_utfSubString := "";

				brwcsncpy(ADR(_utfSubString), _GetNextSubstring.pUtfCsvSubstring, MIN(_GetNextSubstring.Length, 63));
				brwcsconv(ADR(_sSubString), ADR(_utfSubString), 1);
				_diNum := atoi(ADR(_sSubString) );

				CsvStringRow.wArrIdx4 := DINT_TO_UINT(LIMIT(0, _diNum, 65535));

			END_IF

			// Machine Sub Type
			IF NOT _GetNextSubstring.EndOfLine THEN

				_GetNextSubstring(pUtfCsvString := _pUtfCsvString);

				brwcsncpy(ADR(CsvStringRow.utfMachineSubType), _GetNextSubstring.pUtfCsvSubstring, MIN(_GetNextSubstring.Length, 11));

			END_IF

		ELSIF _diRowType = MNPARAM_CSV_DAT_NUM OR _diRowType = MNPARAM_CSV_DAT_REAL THEN

			// CSV Num Parameter
			RowType := DINT_TO_UINT(_diRowType);

			CsvNumRow.bRowType := UINT_TO_USINT(RowType - MNPARAM_CSV_DAT_NUM);

			// Index
			IF NOT _GetNextSubstring.EndOfLine THEN

				_GetNextSubstring(pUtfCsvString := _pUtfCsvString);

				_utfSubString := "";

				brwcsncpy(ADR(_utfSubString), _GetNextSubstring.pUtfCsvSubstring, MIN(_GetNextSubstring.Length, 63));
				brwcsconv(ADR(_sSubString), ADR(_utfSubString), 1);
				_diNum := atoi(ADR(_sSubString) );

				CsvNumRow.wIdxNumPar := DINT_TO_UINT(LIMIT(0, _diNum, 65535));

			END_IF

			IF RowType = 10 THEN

				// Value Integer
				IF NOT _GetNextSubstring.EndOfLine THEN

					_GetNextSubstring(pUtfCsvString := _pUtfCsvString);

					_utfSubString := "";

					brwcsncpy(ADR(_utfSubString), _GetNextSubstring.pUtfCsvSubstring, MIN(_GetNextSubstring.Length, 63));
					brwcsconv(ADR(_sSubString), ADR(_utfSubString), 1);
					CsvNumRow.diValue := atoi(ADR(_sSubString) );

				END_IF

			ELSE

				// Value Real
				IF NOT _GetNextSubstring.EndOfLine THEN

					_GetNextSubstring(pUtfCsvString := _pUtfCsvString);

					_utfSubString := "";

					brwcsncpy(ADR(_utfSubString), _GetNextSubstring.pUtfCsvSubstring, MIN(_GetNextSubstring.Length, 63));
					brwcsconv(ADR(_sSubString), ADR(_utfSubString), 1);
					_rValue := atof(ADR(_sSubString));
					_pdiValue ACCESS ADR(_rValue);
					CsvNumRow.diValue := _pdiValue;

				END_IF

			END_IF

			//  ArrIndex1
			IF NOT _GetNextSubstring.EndOfLine THEN

				_GetNextSubstring(pUtfCsvString := _pUtfCsvString);

				_utfSubString := "";

				brwcsncpy(ADR(_utfSubString), _GetNextSubstring.pUtfCsvSubstring, MIN(_GetNextSubstring.Length, 63));
				brwcsconv(ADR(_sSubString), ADR(_utfSubString), 1);
				_diNum := atoi(ADR(_sSubString) );

				CsvNumRow.wArrIdx1 := DINT_TO_UINT(LIMIT(0, _diNum, 65535));

			END_IF

			//  ArrIndex2
			IF NOT _GetNextSubstring.EndOfLine THEN

				_GetNextSubstring(pUtfCsvString := _pUtfCsvString);

				_utfSubString := "";

				brwcsncpy(ADR(_utfSubString), _GetNextSubstring.pUtfCsvSubstring, MIN(_GetNextSubstring.Length, 63));
				brwcsconv(ADR(_sSubString), ADR(_utfSubString), 1);
				_diNum := atoi(ADR(_sSubString) );

				CsvNumRow.wArrIdx2 := DINT_TO_UINT(LIMIT(0, _diNum, 65535));

			END_IF

			//  ArrIndex3
			IF NOT _GetNextSubstring.EndOfLine THEN

				_GetNextSubstring(pUtfCsvString := _pUtfCsvString);

				_utfSubString := "";

				brwcsncpy(ADR(_utfSubString), _GetNextSubstring.pUtfCsvSubstring, MIN(_GetNextSubstring.Length, 63));
				brwcsconv(ADR(_sSubString), ADR(_utfSubString), 1);
				_diNum := atoi(ADR(_sSubString) );

				CsvNumRow.wArrIdx3 := DINT_TO_UINT(LIMIT(0, _diNum, 65535));

			END_IF

			//  ArrIndex4
			IF NOT _GetNextSubstring.EndOfLine THEN

				_GetNextSubstring(pUtfCsvString := _pUtfCsvString);

				_utfSubString := "";

				brwcsncpy(ADR(_utfSubString), _GetNextSubstring.pUtfCsvSubstring, MIN(_GetNextSubstring.Length, 63));
				brwcsconv(ADR(_sSubString), ADR(_utfSubString), 1);
				_diNum := atoi(ADR(_sSubString) );

				CsvNumRow.wArrIdx4 := DINT_TO_UINT(LIMIT(0, _diNum, 65535));

			END_IF

			// Machine Sub Type
			IF NOT _GetNextSubstring.EndOfLine THEN

				_GetNextSubstring(pUtfCsvString := _pUtfCsvString);

				brwcsncpy(ADR(CsvNumRow.utfMachineSubType), _GetNextSubstring.pUtfCsvSubstring, MIN(_GetNextSubstring.Length, 11));

			END_IF

		END_IF

	ELSE

		status := ERR_FUB_ENABLE_FALSE;

	END_IF

END_FUNCTION_BLOCK
```

#### mnParam_atodatetime.st - String mit ISO-Zeitformat in DATE_AND_TIME wandeln
```iecst
(********************************************************************
 * COPYRIGHT -- Microsoft
 ********************************************************************
 * Library: mnParamLib
 * File: mnParam_atodatetime.st
 * Author: hunholz
 * Created: July 25, 2011
 ********************************************************************
 * Implementation of library mnParamLib
 ********************************************************************)

(* String mit ISO-Zeitformat in DATE_AND_TIME wandeln *)
FUNCTION_BLOCK mnParam_atodatetime

	brsmemset(ADR(dtTimeStamp), 0, SIZEOF(dtTimeStamp));
	brsmemset(ADR(_DateTime), 0, SIZEOF(_DateTime));
	brsmemset(ADR(_sStr), 0, SIZEOF(_sStr));

	IF brsstrlen(pStr) > 23 THEN
		// String abschneiden
		brsmemcpy(ADR(_sStr), pStr, 23);
	ELSE
		brsstrcpy(ADR(_sStr), pStr);
	END_IF

	_wPositionInTime := 0;

	_wPositionInTime := FIND(_sStr, '-');
	IF (_wPositionInTime < 8) THEN
		_sSubString := LEFT(_sStr, _wPositionInTime);
		_DateTime.year := DINT_TO_UINT(atoi(ADR(_sSubString)));
	END_IF

	_sStr := DELETE(_sStr, _wPositionInTime, 1);

	_wPositionInTime := FIND(_sStr, '-');
	IF (_wPositionInTime < 8) THEN
		_sSubString := LEFT(_sStr, _wPositionInTime);
		_DateTime.month := DINT_TO_USINT(atoi(ADR(_sSubString)));
	END_IF

	_sStr := DELETE(_sStr, _wPositionInTime, 1);

	_wPositionInTime := FIND(_sStr, 'T');
	IF (_wPositionInTime < 8) THEN
		_sSubString := LEFT(_sStr, _wPositionInTime);
		_DateTime.day := DINT_TO_USINT(atoi(ADR(_sSubString)));
	END_IF

	_sStr := DELETE(_sStr, _wPositionInTime, 1);

	_wPositionInTime := FIND(_sStr, ':');
	IF (_wPositionInTime < 8) THEN
		_sSubString := LEFT(_sStr, _wPositionInTime);
		_DateTime.hour := DINT_TO_USINT(atoi(ADR(_sSubString)));
	END_IF

	_sStr := DELETE(_sStr, _wPositionInTime, 1);

	_wPositionInTime := FIND(_sStr, ':');
	IF (_wPositionInTime < 8) THEN
		_sSubString := LEFT(_sStr, _wPositionInTime);
		_DateTime.minute := DINT_TO_USINT(atoi(ADR(_sSubString)));
	END_IF

	_sStr := DELETE(_sStr, _wPositionInTime, 1);

	_DateTime.second := DINT_TO_USINT(atoi(ADR(_sStr)));

	IF _DateTime.day = 0 OR _DateTime.month = 0 OR _DateTime.year = 0 THEN

		status := 1;

	ELSE

		dtTimeStamp := DTStructure_TO_DT(ADR(_DateTime));

	END_IF

END_FUNCTION_BLOCK
```

#### mnParam_GetNextSubstring.st
```iecst
(********************************************************************
 * COPYRIGHT -- Microsoft
 ********************************************************************
 * Library: mnParamLib
 * File: mnParam_GetNextSubstring.st
 * Author: hunholz
 * Created: July 26, 2011
 ********************************************************************
 * Implementation of library mnParamLib
 ********************************************************************)

(* TODO: Add your comment here *)
FUNCTION_BLOCK mnParam_GetNextSubstring

	IF enable THEN

		EndOfLine := FALSE;
		brsmemset(ADR(_utfSubString), 0, SIZEOF(_utfSubString));

		// Länge des Strings ermitteln
		_lLen :=  brwcslen(pUtfCsvString);

		// Tab-Zeichen suchen
		_lAdrTab := brwcschr(pUtfCsvString, 16#0009);

		// Kein Tab-Zeichen gefunden, dann String zurückgeben und EndOfLine auf TRUE setzen
		IF _lAdrTab = 0 THEN

			EndOfLine := TRUE;
			Length := MIN(255,_lLen);
			brwcsncpy(ADR(_utfSubString), pUtfCsvString, Length);

		ELSE

			_lLen := (_lAdrTab - pUtfCsvString ) / 2;
			Length := MIN(255, _lLen);
			IF Length = 0 THEN
				_utfSubString := "";
			ELSE
				brwcsncpy(ADR(_utfSubString), pUtfCsvString, Length);
			END_IF
			pUtfCsvString := _lAdrTab + 2;

		END_IF

		pUtfCsvSubstring := ADR(_utfSubString);

		status := ERR_OK;

	ELSE

		status := ERR_FUB_ENABLE_FALSE;

	END_IF

END_FUNCTION_BLOCK
```

#### mnParam_GetContainerOfParamNum.st - ContainerID ermitteln und Array-Grenzen
```iecst
(********************************************************************
 * COPYRIGHT -- Microsoft
 ********************************************************************
 * Library: mnParamLib
 * File: mnParam_GetContainerOfParamNum.st
 * Author: hunholz
 * Created: July 27, 2011
 ********************************************************************
 * Implementation of library mnParamLib
 ********************************************************************)

(* ContainerID ermitteln und Array-Grenzen *)
FUNCTION_BLOCK mnParam_GetContainerOfParamNum

	IF enable THEN

		status := 0;
		brsmemset(ADR(wMinBound), 0, SIZEOF(wMinBound));
		brsmemset(ADR(wDimension), 0, SIZEOF(wDimension));
		wCountArray := 0;
		iContainer := 127;

		IF pLogicStructs = 0 OR pParamNum = 0 THEN

			status := 1;
			RETURN;

		END_IF

		_LS ACCESS pLogicStructs;
		_PN ACCESS pParamNum;

		IF _PN.wReferenz = 0 OR _PN.wReferenz > wMaxIdxLogicStructs THEN

			status := 2;
			RETURN;

		END_IF

		_bMaxCycle := 0;
		_iIdxLS := UINT_TO_INT(_PN.wReferenz);

		IF _PN.wDimension > 0 THEN
			wCountArray := 1;
			wDimension[1] := _PN.wDimension;
			wMinBound[1] := _PN.wMinBound;
		END_IF

		IF _LS[_iIdxLS].wDimension > 0 THEN

			wCountArray := wCountArray + 1;

			IF wCountArray > 1 THEN
				FOR _i := 2 TO wCountArray DO
					wDimension[wCountArray - _i + 2] := wDimension[wCountArray - _i + 1];
					wMinBound[wCountArray - _i + 2] := wMinBound[wCountArray - _i + 1];
				END_FOR
			END_IF

			wDimension[1] := _LS[_iIdxLS].wDimension;
			wMinBound[1] := _LS[_iIdxLS].wMinBound;

		END_IF

		REPEAT

			IF _LS[_iIdxLS].iReferenz > 0 THEN

				IF INT_TO_UINT(_LS[_iIdxLS].iReferenz) > wMaxIdxLogicStructs THEN
					status := 10;
					RETURN;
				END_IF

				_iIdxLS := _LS[_iIdxLS].iReferenz;

				IF _LS[_iIdxLS].wDimension > 0 THEN

					IF wCountArray >= 4 THEN
						status := 3;
						RETURN;
					END_IF

					wCountArray := wCountArray + 1;

					IF wCountArray > 1 THEN
						FOR _i := 2 TO wCountArray DO
							wDimension[wCountArray - _i + 2] := wDimension[wCountArray - _i + 1];
							wMinBound[wCountArray - _i + 2] := wMinBound[wCountArray - _i + 1];
						END_FOR
					END_IF

					wDimension[1] := _LS[_iIdxLS].wDimension;
					wMinBound[1] := _LS[_iIdxLS].wMinBound;

				END_IF

				_bMaxCycle := _bMaxCycle + 1;

			END_IF

			IF _bMaxCycle >= 30 THEN
				status := 4;
				RETURN;
			END_IF

			IF _LS[_iIdxLS].iReferenz <= 0 THEN
				iContainer := _LS[_iIdxLS].iReferenz;
				RETURN;
			END_IF

		UNTIL
			FALSE
		END_REPEAT

	ELSE

		status := ERR_FUB_ENABLE_FALSE;

	END_IF

END_FUNCTION_BLOCK
```

#### mnParam_GetContainerOfParamStrin.st - Container für String-Parameter bestimmen
```iecst
(********************************************************************
 * COPYRIGHT -- Microsoft
 ********************************************************************
 * Library: mnParamLib
 * File: mnParam_GetContainerOfParamStrin.st
 * Author: hunholz
 * Created: July 27, 2011
 ********************************************************************
 * Implementation of library mnParamLib
 ********************************************************************)

(* Container für String-Parameter bestimmen *)
FUNCTION_BLOCK mnParam_GetContainerOfParamStrin

	IF enable THEN

		status := 0;
		brsmemset(ADR(wMinBound), 0, SIZEOF(wMinBound));
		brsmemset(ADR(wDimension), 0, SIZEOF(wDimension));
		wCountArray := 0;
		iContainer := 127;

		IF pLogicStructs = 0 OR pParamString = 0 THEN

			status := 1;
			RETURN;

		END_IF

		_LS ACCESS pLogicStructs;
		_PS ACCESS pParamString;

		IF _PS.wReferenz = 0 OR _PS.wReferenz > wMaxIdxLogicStructs THEN

			status := 2;
			RETURN;

		END_IF

		_bMaxCycle := 0;
		_iIdxLS := UINT_TO_INT(_PS.wReferenz);

		IF _PS.wDimension > 0 THEN
			wCountArray := 1;
			wDimension[1] := _PS.wDimension;
			wMinBound[1] := _PS.wMinBound;
		END_IF

		IF _LS[_iIdxLS].wDimension > 0 THEN

			wCountArray := wCountArray + 1;

			IF wCountArray > 1 THEN
				FOR _i := 2 TO wCountArray DO
					wDimension[wCountArray - _i + 2] := wDimension[wCountArray - _i + 1];
					wMinBound[wCountArray - _i + 2] := wMinBound[wCountArray - _i + 1];
				END_FOR
			END_IF

			wDimension[1] := _LS[_iIdxLS].wDimension;
			wMinBound[1] := _LS[_iIdxLS].wMinBound;

		END_IF

		REPEAT

			IF _LS[_iIdxLS].iReferenz > 0 THEN

				IF INT_TO_UINT(_LS[_iIdxLS].iReferenz) > wMaxIdxLogicStructs THEN
					status := 10;
					RETURN;
				END_IF

				_iIdxLS := _LS[_iIdxLS].iReferenz;

				IF _LS[_iIdxLS].wDimension > 0 THEN

					IF wCountArray >= 4 THEN
						status := 3;
						RETURN;
					END_IF

					wCountArray := wCountArray + 1;

					IF wCountArray > 1 THEN
						FOR _i := 2 TO wCountArray DO
							wDimension[wCountArray - _i + 2] := wDimension[wCountArray - _i + 1];
							wMinBound[wCountArray - _i + 2] := wMinBound[wCountArray - _i + 1];
						END_FOR
					END_IF

					wDimension[1] := _LS[_iIdxLS].wDimension;
					wMinBound[1] := _LS[_iIdxLS].wMinBound;

				END_IF

				_bMaxCycle := _bMaxCycle + 1;

			END_IF

			IF _bMaxCycle >= 30 THEN
				status := 4;
				RETURN;
			END_IF

			IF _LS[_iIdxLS].iReferenz <= 0 THEN
				iContainer := (_LS[_iIdxLS].iReferenz);
				RETURN;
			END_IF

		UNTIL
			FALSE
		END_REPEAT

	ELSE

		status := ERR_FUB_ENABLE_FALSE;

	END_IF

END_FUNCTION_BLOCK
```

#### GetArrayPV.st - Liefert PV-Adresse mit Indizes
```iecst
(********************************************************************
 * COPYRIGHT -- Microsoft
 ********************************************************************
 * Library: mnParamLib
 * File: GetArrayPV.st
 * Author: hunholz
 * Created: July 27, 2011
 ********************************************************************
 * Implementation of library mnParamLib
 ********************************************************************)

(* Liefert PV-Adresse mit Indizes *)
FUNCTION GetArrayPV

	GetArrayPV := 0;

	IF pPV = 0  OR pPVFilled = 0 OR pStructRoot = 0 THEN
		GetArrayPV := 1;
		RETURN;
	END_IF

	_GetArrayPV ACCESS pPVFilled;
	_GetArrayPV := '';

	brsstrcpy(pPVFilled, pStructRoot);
	brsstrcat(pPVFilled, pPV);

	_p := FIND(_GetArrayPV, '[]') ;
	IF _p <> 0 THEN
		brsitoa(idx1, ADR(_sIndex));
		_GetArrayPV := INSERT(_GetArrayPV, _sIndex, _p);
		_p := FIND(_GetArrayPV, '[]') ;
		IF _p <> 0 THEN
			brsitoa(idx2, ADR(_sIndex));
			_GetArrayPV := INSERT(_GetArrayPV, _sIndex, _p);
			_p := FIND(_GetArrayPV, '[]') ;
			IF _p <> 0 THEN
				brsitoa(idx3, ADR(_sIndex));
				_GetArrayPV := INSERT(_GetArrayPV, _sIndex, _p);
				_p := FIND(_GetArrayPV, '[]') ;
				IF _p <> 0 THEN
					brsitoa(idx4, ADR(_sIndex));
					_GetArrayPV := INSERT(_GetArrayPV, _sIndex, _p);
				END_IF
			END_IF
		END_IF
	END_IF

END_FUNCTION
```

#### mnParam_WritePVNum.st - DINT auf beliebige, numerische Variable schreiben
```iecst
(********************************************************************
 * COPYRIGHT -- Microsoft
 ********************************************************************
 * Library: mnParamLib
 * File: mnParam_WritePVNum.st
 * Author: hunholz
 * Created: July 27, 2011
 * Changed: November 28, 2011
 * ###AH20111128 DINT_TO_UINT gegen DINT_TO_UDINT getauscht. UDINT wurde abgeschnitten.
 ********************************************************************
 * Implementation of library mnParamLib
 ********************************************************************)

(* DINT auf beliebige, numerische Variable schreiben *)
FUNCTION_BLOCK mnParam_WritePVNum

	status := 0;

	IF pAdress = 0 THEN
		status := 1;
		RETURN;
	END_IF

	status := PV_xgetadr(pAdress, ADR(_lPVadress), ADR(_lPVlen));

	IF status = ERR_OK THEN

		status := PV_ninfo(pAdress, ADR(_lPVdataType), ADR(_lDataLen),  ADR(_wDataDimension));

		IF  status = ERR_OK THEN

			IF _lPVdataType = 1 THEN
				// Bool
				_pBool ACCESS _lPVadress;
				_pBool := DINT_TO_BOOL(LIMIT(0, diValue ,1));
			ELSIF _lPVdataType = 2 THEN
				// SINT
				_pSint ACCESS _lPVadress;
				_pSint := DINT_TO_SINT(LIMIT(-128, diValue, 127));
			ELSIF _lPVdataType = 3 THEN
				// INT
				_pInt ACCESS _lPVadress;
				_pInt := DINT_TO_INT(LIMIT(-32768, diValue, 32767));
			ELSIF _lPVdataType = 4 THEN
				// DINT
				_pDint ACCESS _lPVadress;
				_pDint := diValue;
			ELSIF _lPVdataType = 5 THEN
				// USINT
				_pUsint ACCESS _lPVadress;
				_pUsint := DINT_TO_USINT(LIMIT(0,diValue,255));
			ELSIF _lPVdataType = 6 THEN
				// UINT
				_pUint ACCESS _lPVadress;
				_pUint := DINT_TO_UINT(LIMIT(0,diValue,65535));
			ELSIF _lPVdataType = 7 THEN
				// UDINT
				_pUdint ACCESS _lPVadress;
				_pUdint := DINT_TO_UDINT(LIMIT(0,diValue,16#7FFFFFFF));
			ELSIF _lPVdataType = 8 THEN
				// REAL
				_pReal ACCESS _lPVadress;
				_pReal := DINT_TO_REAL(diValue);
			ELSIF _lPVdataType = 11 THEN
				// DATE_AND_TIME
				_pDT ACCESS _lPVadress;
				_pDT := DINT_TO_DT(diValue);
			ELSIF _lPVdataType = 12 THEN
				// TIME
				_pT ACCESS _lPVadress;
				_pT := DINT_TO_TIME(diValue);
			ELSE
				status := 2;
			END_IF

		END_IF

	END_IF

END_FUNCTION_BLOCK
```

#### mnParam_WritePVrNum.st - REAL auf beliebige, numerische Variable schreiben
```iecst
(********************************************************************
 * COPYRIGHT -- Microsoft
 ********************************************************************
 * Library: mnParamLib
 * File: mnParam_WritePVrNum.st
 * Author: hunholz
 * Created: August 18, 2011
 ********************************************************************
 * Implementation of library mnParamLib
 ********************************************************************)

(* REAL auf  numerische Variable schreiben *)
FUNCTION_BLOCK mnParam_WritePVrNum

	status := 0;

	IF pAdress = 0 THEN
		status := 1;
		RETURN;
	END_IF

	status := PV_xgetadr(pAdress, ADR(_lPVadress), ADR(_lPVlen));
	IF status = ERR_OK THEN

		status := PV_ninfo(pAdress, ADR(_lPVdataType), ADR(_lDataLen),  ADR(_wDataDimension));
		IF  status = ERR_OK THEN

			IF _lPVdataType = 8 THEN
				// REAL
				_pReal ACCESS _lPVadress;
				_pReal := rValue;
			ELSE
				status := 2;
			END_IF

		END_IF

	ELSE

	END_IF

END_FUNCTION_BLOCK
```

#### mnParam_WritePVString.st - Schreibe String-Variable
```iecst
(********************************************************************
 * COPYRIGHT -- Microsoft
 ********************************************************************
 * Library: mnParamLib
 * File: mnParam_WritePVString.st
 * Author: hunholz
 * Created: July 27, 2011
 ********************************************************************
 * Implementation of library mnParamLib
 ********************************************************************)

(* Schreibe String-Variable *)
FUNCTION_BLOCK mnParam_WritePVString

	status := 0;

	IF pAdress = 0 OR p_utfValue = 0 THEN
		status := 1;
		RETURN;
	END_IF

	status := PV_xgetadr(pAdress, ADR(_lPVadress), ADR(_lPVlen));
	IF status = ERR_OK THEN

		status := PV_ninfo(pAdress, ADR(_lPVdataType), ADR(_lDataLen),  ADR(_wDataDimension));
		IF  status = ERR_OK THEN

			IF _lPVdataType = 6 THEN

				// UINT-Array für utf-Strings

				brwcsncpy(_lPVadress, p_utfValue, _wDataDimension-1);

			ELSIF _lPVdataType = 9 THEN

				// STRING
				brsmemset(_lPVadress, 0, _lPVlen);

				brwcsncpy(ADR(_utfValue), p_utfValue, MIN(31, _lPVlen-1));
				brwcsconv(_lPVadress, ADR(_utfValue), 1);

			ELSIF _lPVdataType = 21 THEN

				// WSTRING
				brsmemset(_lPVadress, 0, _lPVlen);

				brwcsncpy(_lPVadress, p_utfValue, MIN(31, (_lPVlen/2)-1));

			ELSE

				status := 2;

			END_IF
		END_IF
	END_IF

END_FUNCTION_BLOCK
```

#### mnParam_WriteBOM_Mem.st - Byte Order Mark
```iecst
(********************************************************************
 * COPYRIGHT -- Microsoft
 ********************************************************************
 * Library: mnParamLib
 * File: mnParam_WriteBOM_Mem.st
 * Author: hunholz
 * Created: August 01, 2011
 ********************************************************************
 * Implementation of library mnParamLib
 ********************************************************************)

(* Byte Order Mark *)
FUNCTION_BLOCK mnParam_WriteBOM_Mem

	IF enable THEN

		IF pMem = 0 THEN

			status := 1;
			RETURN;

		END_IF

		IF (lSize + 2) <= lMaxSize THEN

			_pUtfString ACCESS pMem;

			_pUtfString := 16#FEFF;	// BOM

			lSize := lSize + 2;

		ELSE

			status := 2;
			RETURN;

		END_IF

		status := 0;

	ELSE

		status := 65334;

	END_IF

END_FUNCTION_BLOCK
```

#### mnParam_WriteNewline_Mem.st - Leerzeile
```iecst
(********************************************************************
 * COPYRIGHT -- Microsoft
 ********************************************************************
 * Library: mnParamLib
 * File: mnParam_WriteNewline_Mem.st
 * Author: hunholz
 * Created: August 02, 2011
 ********************************************************************
 * Implementation of library mnParamLib
 ********************************************************************)

(* Leerzeile *)
FUNCTION_BLOCK mnParam_WriteNewline_Mem

	IF enable THEN

		IF pMem = 0 THEN

			status := 1;
			RETURN;

		END_IF

		IF (lSize + 4) <= lMaxSize THEN

			_pUtfString ACCESS pMem + lSize;

			_pUtfString[0] := 16#000D;	// Return
			_pUtfString[1] := 16#000A;	// Newline

			lSize := lSize + 4;

		ELSE

			status := 2;
			RETURN;

		END_IF

		status := 0;

	ELSE

		status := 65334;

	END_IF
END_FUNCTION_BLOCK
```

#### mnParam_WriteCSV10_Mem.st - Datenzeile numerisch schreiben
```iecst
(********************************************************************
 * COPYRIGHT -- Microsoft
 ********************************************************************
 * Library: mnParamLib
 * File: mnParam_WriteCSV10_Mem.st
 * Author: hunholz
 * Created: August 02, 2011
 ********************************************************************
 * Implementation of library mnParamLib
 ********************************************************************)

(* Datenzeile numerisch schreiben *)
FUNCTION_BLOCK mnParam_WriteCSV10_Mem

	IF enable THEN

		IF pMem = 0 THEN

			status := 1;
			RETURN;

		END_IF

		IF (lSize + 6) <= lMaxSize THEN

			_pUtfString ACCESS pMem + lSize;

			_pUtfString[0] := 16#0031;	// 1
			_pUtfString[1] := 16#0030;	// 0
			_pUtfString[2] := 16#0009;	// TAB

			lSize := lSize + 6;

		ELSE

			status := 2;
			RETURN;

		END_IF

		// IdxNumPar schreiben

		brsitoa(NumRow.wIdxNumPar, ADR(_sNumeric));

		_lLen := LEN(_sNumeric);

		IF _lLen > 0 THEN

			IF (lSize + _lLen*2 ) <= lMaxSize THEN

				brwcsconv(pMem + lSize, ADR(_sNumeric), 0);

				lSize := lSize + 2* _lLen;

			ELSE

				status := 2;
				RETURN;

			END_IF

		END_IF

		IF (lSize + 2) <= lMaxSize THEN

			_pUtfString ACCESS pMem + lSize;

			_pUtfString[0] := 16#0009;	// TAB

			lSize := lSize + 2;

		ELSE

			status := 2;
			RETURN;

		END_IF

		// Value schreiben

		brsitoa(NumRow.diValue, ADR(_sNumeric));

		_lLen := LEN(_sNumeric);

		IF _lLen > 0 THEN

			IF (lSize + _lLen*2 ) <= lMaxSize THEN

				brwcsconv(pMem + lSize, ADR(_sNumeric), 0);

				lSize := lSize + 2* _lLen;

			ELSE

				status := 2;
				RETURN;

			END_IF

		END_IF

		IF (lSize + 2) <= lMaxSize THEN

			_pUtfString ACCESS pMem + lSize;

			_pUtfString[0] := 16#0009;	// TAB

			lSize := lSize + 2;

		ELSE

			status := 2;
			RETURN;

		END_IF

		// 1 Array Index

		brsitoa(NumRow.wArrIdx1, ADR(_sNumeric));

		_lLen := LEN(_sNumeric);

		IF _lLen > 0 THEN

			IF (lSize + _lLen*2 ) <= lMaxSize THEN

				brwcsconv(pMem + lSize, ADR(_sNumeric), 0);

				lSize := lSize + 2* _lLen;

			ELSE

				status := 2;
				RETURN;

			END_IF

		END_IF

		IF (lSize + 2) <= lMaxSize THEN

			_pUtfString ACCESS pMem + lSize;

			_pUtfString[0] := 16#0009;	// TAB

			lSize := lSize + 2;

		ELSE

			status := 2;
			RETURN;

		END_IF

		// 2 Array Index

		brsitoa(NumRow.wArrIdx2, ADR(_sNumeric));

		_lLen := LEN(_sNumeric);

		IF _lLen > 0 THEN

			IF (lSize + _lLen*2 ) <= lMaxSize THEN

				brwcsconv(pMem + lSize, ADR(_sNumeric), 0);

				lSize := lSize + 2* _lLen;

			ELSE

				status := 2;
				RETURN;

			END_IF

		END_IF

		IF (lSize + 2) <= lMaxSize THEN

			_pUtfString ACCESS pMem + lSize;

			_pUtfString[0] := 16#0009;	// TAB

			lSize := lSize + 2;

		ELSE

			status := 2;
			RETURN;

		END_IF

		// 3 Array Index

		brsitoa(NumRow.wArrIdx3, ADR(_sNumeric));

		_lLen := LEN(_sNumeric);

		IF _lLen > 0 THEN

			IF (lSize + _lLen*2 ) <= lMaxSize THEN

				brwcsconv(pMem + lSize, ADR(_sNumeric), 0);

				lSize := lSize + 2* _lLen;

			ELSE

				status := 2;
				RETURN;

			END_IF

		END_IF

		IF (lSize + 2) <= lMaxSize THEN

			_pUtfString ACCESS pMem + lSize;

			_pUtfString[0] := 16#0009;	// TAB

			lSize := lSize + 2;

		ELSE

			status := 2;
			RETURN;

		END_IF

		// 4 Array Index

		brsitoa(NumRow.wArrIdx4, ADR(_sNumeric));

		_lLen := LEN(_sNumeric);

		IF _lLen > 0 THEN

			IF (lSize + _lLen*2 ) <= lMaxSize THEN

				brwcsconv(pMem + lSize, ADR(_sNumeric), 0);

				lSize := lSize + 2* _lLen;

			ELSE

				status := 2;
				RETURN;

			END_IF

		END_IF

		IF (lSize + 2) <= lMaxSize THEN

			_pUtfString ACCESS pMem + lSize;

			_pUtfString[0] := 16#0009;	// TAB

			lSize := lSize + 2;

		ELSE

			status := 2;
			RETURN;

		END_IF

		// Maschinensubtyp schreiben

		_lLen := brwcslen(ADR(NumRow.utfMachineSubType));

		IF _lLen > 0 THEN

			IF (lSize + _lLen*2 ) <= lMaxSize THEN

				brwcscpy(pMem + lSize, ADR(NumRow.utfMachineSubType));

				lSize := lSize + 2* _lLen;

			ELSE

				status := 2;
				RETURN;

			END_IF

		END_IF

		IF (lSize + 4) <= lMaxSize THEN

			_pUtfString ACCESS pMem + lSize;

			_pUtfString[0] := 16#000D;	// Return
			_pUtfString[1] := 16#000A;	// Linefeed

			lSize := lSize + 4;

		ELSE

			status := 2;
			RETURN;

		END_IF

		status := 0;

	ELSE

		status := 65334;

	END_IF

END_FUNCTION_BLOCK
```

#### mnParam_WriteCSV11_Mem.st - Datenzeile numerisch schreiben
```iecst
(********************************************************************
 * COPYRIGHT -- Microsoft
 ********************************************************************
 * Library: mnParamLib
 * File: mnParam_WriteCSV11_Mem.st
 * Author: hunholz
 * Created: August 18, 2011
 ********************************************************************
 * Implementation of library mnParamLib
 ********************************************************************)

(* Datenzeile numerisch schreiben *)
FUNCTION_BLOCK mnParam_WriteCSV11_Mem

	IF enable THEN

		IF pMem = 0 THEN

			status := 1;
			RETURN;

		END_IF

		IF (lSize + 6) <= lMaxSize THEN

			_pUtfString ACCESS pMem + lSize;

			_pUtfString[0] := 16#0031;	// 1
			_pUtfString[1] := 16#0031;	// 1
			_pUtfString[2] := 16#0009;	// TAB

			lSize := lSize + 6;

		ELSE

			status := 2;
			RETURN;

		END_IF

		// IdxNumPar schreiben

		brsitoa(NumRow.wIdxNumPar, ADR(_sNumeric));

		_lLen := LEN(_sNumeric);

		IF _lLen > 0 THEN

			IF (lSize + _lLen*2 ) <= lMaxSize THEN

				brwcsconv(pMem + lSize, ADR(_sNumeric), 0);

				lSize := lSize + 2* _lLen;

			ELSE

				status := 2;
				RETURN;

			END_IF

		END_IF

		IF (lSize + 2) <= lMaxSize THEN

			_pUtfString ACCESS pMem + lSize;

			_pUtfString[0] := 16#0009;	// TAB

			lSize := lSize + 2;

		ELSE

			status := 2;
			RETURN;

		END_IF

		// Value schreiben

		_pdiValue ACCESS ADR(_rValue);
		_pdiValue := NumRow.diValue;
		brsftoa(_rValue, ADR(_sNumeric));

		_lLen := LEN(_sNumeric);

		IF _lLen > 0 THEN

			IF (lSize + _lLen*2 ) <= lMaxSize THEN

				brwcsconv(pMem + lSize, ADR(_sNumeric), 0);

				lSize := lSize + 2* _lLen;

			ELSE

				status := 2;
				RETURN;

			END_IF

		END_IF

		IF (lSize + 2) <= lMaxSize THEN

			_pUtfString ACCESS pMem + lSize;

			_pUtfString[0] := 16#0009;	// TAB

			lSize := lSize + 2;

		ELSE

			status := 2;
			RETURN;

		END_IF

		// 1 Array Index

		brsitoa(NumRow.wArrIdx1, ADR(_sNumeric));

		_lLen := LEN(_sNumeric);

		IF _lLen > 0 THEN

			IF (lSize + _lLen*2 ) <= lMaxSize THEN

				brwcsconv(pMem + lSize, ADR(_sNumeric), 0);

				lSize := lSize + 2* _lLen;

			ELSE

				status := 2;
				RETURN;

			END_IF

		END_IF

		IF (lSize + 2) <= lMaxSize THEN

			_pUtfString ACCESS pMem + lSize;

			_pUtfString[0] := 16#0009;	// TAB

			lSize := lSize + 2;

		ELSE

			status := 2;
			RETURN;

		END_IF

		// 2 Array Index

		brsitoa(NumRow.wArrIdx2, ADR(_sNumeric));

		_lLen := LEN(_sNumeric);

		IF _lLen > 0 THEN

			IF (lSize + _lLen*2 ) <= lMaxSize THEN

				brwcsconv(pMem + lSize, ADR(_sNumeric), 0);

				lSize := lSize + 2* _lLen;

			ELSE

				status := 2;
				RETURN;

			END_IF

		END_IF

		IF (lSize + 2) <= lMaxSize THEN

			_pUtfString ACCESS pMem + lSize;

			_pUtfString[0] := 16#0009;	// TAB

			lSize := lSize + 2;

		ELSE

			status := 2;
			RETURN;

		END_IF

		// 3 Array Index

		brsitoa(NumRow.wArrIdx3, ADR(_sNumeric));

		_lLen := LEN(_sNumeric);

		IF _lLen > 0 THEN

			IF (lSize + _lLen*2 ) <= lMaxSize THEN

				brwcsconv(pMem + lSize, ADR(_sNumeric), 0);

				lSize := lSize + 2* _lLen;

			ELSE

				status := 2;
				RETURN;

			END_IF

		END_IF

		IF (lSize + 2) <= lMaxSize THEN

			_pUtfString ACCESS pMem + lSize;

			_pUtfString[0] := 16#0009;	// TAB

			lSize := lSize + 2;

		ELSE

			status := 2;
			RETURN;

		END_IF

		// 4 Array Index

		brsitoa(NumRow.wArrIdx4, ADR(_sNumeric));

		_lLen := LEN(_sNumeric);

		IF _lLen > 0 THEN

			IF (lSize + _lLen*2 ) <= lMaxSize THEN

				brwcsconv(pMem + lSize, ADR(_sNumeric), 0);

				lSize := lSize + 2* _lLen;

			ELSE

				status := 2;
				RETURN;

			END_IF

		END_IF

		IF (lSize + 2) <= lMaxSize THEN

			_pUtfString ACCESS pMem + lSize;

			_pUtfString[0] := 16#0009;	// TAB

			lSize := lSize + 2;

		ELSE

			status := 2;
			RETURN;

		END_IF

		// Maschinensubtyp schreiben

		_lLen := brwcslen(ADR(NumRow.utfMachineSubType));

		IF _lLen > 0 THEN

			IF (lSize + _lLen*2 ) <= lMaxSize THEN

				brwcscpy(pMem + lSize, ADR(NumRow.utfMachineSubType));

				lSize := lSize + 2* _lLen;

			ELSE

				status := 2;
				RETURN;

			END_IF

		END_IF

		IF (lSize + 4) <= lMaxSize THEN

			_pUtfString ACCESS pMem + lSize;

			_pUtfString[0] := 16#000D;	// Return
			_pUtfString[1] := 16#000A;	// Linefeed

			lSize := lSize + 4;

		ELSE

			status := 2;
			RETURN;

		END_IF

		status := 0;

	ELSE

		status := 65334;

	END_IF

END_FUNCTION_BLOCK
```

#### mnParam_WriteCSV20_Mem.st - String Daten schreiben
```iecst
(********************************************************************
 * COPYRIGHT -- Microsoft
 ********************************************************************
 * Library: mnParamLib
 * File: mnParam_WriteCSV20_Mem.st
 * Author: hunholz
 * Created: August 02, 2011
 ********************************************************************
 * Implementation of library mnParamLib
 ********************************************************************)

(* String Daten schreiben *)
FUNCTION_BLOCK mnParam_WriteCSV20_Mem

	IF enable THEN

		IF pMem = 0 THEN

			status := 1;
			RETURN;

		END_IF

		IF (lSize + 6) <= lMaxSize THEN

			_pUtfString ACCESS pMem + lSize;

			_pUtfString[0] := 16#0032;	// 2
			_pUtfString[1] := 16#0030;	// 0
			_pUtfString[2] := 16#0009;	// TAB

			lSize := lSize + 6;

		ELSE

			status := 2;
			RETURN;

		END_IF

		// IdxNumPar schreiben

		brsitoa(StringRow.wIdxStringPar, ADR(_sNumeric));

		_lLen := LEN(_sNumeric);

		IF _lLen > 0 THEN

			IF (lSize + _lLen*2 ) <= lMaxSize THEN

				brwcsconv(pMem + lSize, ADR(_sNumeric), 0);

				lSize := lSize + 2* _lLen;

			ELSE

				status := 2;
				RETURN;

			END_IF

		END_IF

		IF (lSize + 2) <= lMaxSize THEN

			_pUtfString ACCESS pMem + lSize;

			_pUtfString[0] := 16#0009;	// TAB

			lSize := lSize + 2;

		ELSE

			status := 2;
			RETURN;

		END_IF

		// Value schreiben

		_lLen := brwcslen(ADR(StringRow.utfValue));

		IF _lLen > 0 THEN

			IF (lSize + _lLen*2 ) <= lMaxSize THEN

				brwcscpy(pMem + lSize, ADR(StringRow.utfValue));

				lSize := lSize + 2* _lLen;

			ELSE

				status := 2;
				RETURN;

			END_IF

		END_IF

		IF (lSize + 2) <= lMaxSize THEN

			_pUtfString ACCESS pMem + lSize;

			_pUtfString[0] := 16#0009;	// TAB

			lSize := lSize + 2;

		ELSE

			status := 2;
			RETURN;

		END_IF

		// 1 Array Index

		brsitoa(StringRow.wArrIdx1, ADR(_sNumeric));

		_lLen := LEN(_sNumeric);

		IF _lLen > 0 THEN

			IF (lSize + _lLen*2 ) <= lMaxSize THEN

				brwcsconv(pMem + lSize, ADR(_sNumeric), 0);

				lSize := lSize + 2* _lLen;

			ELSE

				status := 2;
				RETURN;

			END_IF

		END_IF

		IF (lSize + 2) <= lMaxSize THEN

			_pUtfString ACCESS pMem + lSize;

			_pUtfString[0] := 16#0009;	// TAB

			lSize := lSize + 2;

		ELSE

			status := 2;
			RETURN;

		END_IF

		// 2 Array Index

		brsitoa(StringRow.wArrIdx2, ADR(_sNumeric));

		_lLen := LEN(_sNumeric);

		IF _lLen > 0 THEN

			IF (lSize + _lLen*2 ) <= lMaxSize THEN

				brwcsconv(pMem + lSize, ADR(_sNumeric), 0);

				lSize := lSize + 2* _lLen;

			ELSE

				status := 2;
				RETURN;

			END_IF

		END_IF

		IF (lSize + 2) <= lMaxSize THEN

			_pUtfString ACCESS pMem + lSize;

			_pUtfString[0] := 16#0009;	// TAB

			lSize := lSize + 2;

		ELSE

			status := 2;
			RETURN;

		END_IF

		// 3 Array Index

		brsitoa(StringRow.wArrIdx3, ADR(_sNumeric));

		_lLen := LEN(_sNumeric);

		IF _lLen > 0 THEN

			IF (lSize + _lLen*2 ) <= lMaxSize THEN

				brwcsconv(pMem + lSize, ADR(_sNumeric), 0);

				lSize := lSize + 2* _lLen;

			ELSE

				status := 2;
				RETURN;

			END_IF

		END_IF

		IF (lSize + 2) <= lMaxSize THEN

			_pUtfString ACCESS pMem + lSize;

			_pUtfString[0] := 16#0009;	// TAB

			lSize := lSize + 2;

		ELSE

			status := 2;
			RETURN;

		END_IF

		// 4 Array Index

		brsitoa(StringRow.wArrIdx4, ADR(_sNumeric));

		_lLen := LEN(_sNumeric);

		IF _lLen > 0 THEN

			IF (lSize + _lLen*2 ) <= lMaxSize THEN

				brwcsconv(pMem + lSize, ADR(_sNumeric), 0);

				lSize := lSize + 2* _lLen;

			ELSE

				status := 2;
				RETURN;

			END_IF

		END_IF

		IF (lSize + 2) <= lMaxSize THEN

			_pUtfString ACCESS pMem + lSize;

			_pUtfString[0] := 16#0009;	// TAB

			lSize := lSize + 2;

		ELSE

			status := 2;
			RETURN;

		END_IF

		// Maschinensubtyp schreiben

		_lLen := brwcslen(ADR(StringRow.utfMachineSubType));

		IF _lLen > 0 THEN

			IF (lSize + _lLen*2 ) <= lMaxSize THEN

				brwcscpy(pMem + lSize, ADR(StringRow.utfMachineSubType));

				lSize := lSize + 2* _lLen;

			ELSE

				status := 2;
				RETURN;

			END_IF

		END_IF

		IF (lSize + 4) <= lMaxSize THEN

			_pUtfString ACCESS pMem + lSize;

			_pUtfString[0] := 16#000D;	// Return
			_pUtfString[1] := 16#000A;	// Linefeed

			lSize := lSize + 4;

		ELSE

			status := 2;
			RETURN;

		END_IF

		status := 0;

	ELSE

		status := 65334;

	END_IF

END_FUNCTION_BLOCK
```

#### mnParam_WriteCSV81_Mem.st - String Daten schreiben
```iecst
(********************************************************************
 * COPYRIGHT -- Microsoft
 ********************************************************************
 * Library: mnParamLib
 * File: mnParam_WriteCSV81_Mem.st
 * Author: hunholz
 * Created: Mar 29, 2012
 ********************************************************************
 * Implementation of library mnParamLib
 ********************************************************************)

(* String Daten schreiben *)
FUNCTION_BLOCK mnParam_WriteCSV81_Mem

	IF enable THEN

		status := ERR_OK;

		IF pMem = 0 THEN

			status := 1;
			RETURN;

		END_IF

		IF (lSize + 6) <= lMaxSize THEN

			_pUtfString ACCESS pMem + lSize;

			_pUtfString[0] := 16#0038;	// 8
			_pUtfString[1] := 16#0031;	// 1
			_pUtfString[2] := 16#0009;	// TAB

			lSize := lSize + 6;

		ELSE

			status := 2;
			RETURN;

		END_IF

		// Category

		_lLen := LEN(CPRow.sCategory);

		IF _lLen > 0 THEN

			IF (lSize + _lLen*2 ) <= lMaxSize THEN

				brwcsconv(pMem + lSize, ADR(CPRow.sCategory), 0);

				lSize := lSize + 2* _lLen;

			ELSE

				status := 2;
				RETURN;

			END_IF

		END_IF

		IF (lSize + 2) <= lMaxSize THEN

			_pUtfString ACCESS pMem + lSize;

			_pUtfString[0] := 16#0009;	// TAB

			lSize := lSize + 2;

		ELSE

			status := 2;
			RETURN;

		END_IF

		// Categoryname schreiben

		_lLen := brwcslen(ADR(CPRow.utfCategoryName));

		IF _lLen > 0 THEN

			IF (lSize + _lLen*2 ) <= lMaxSize THEN

				brwcscpy(pMem + lSize, ADR(CPRow.utfCategoryName));

				lSize := lSize + 2* _lLen;

			ELSE

				status := 2;
				RETURN;

			END_IF

		END_IF

		IF (lSize + 2) <= lMaxSize THEN

			_pUtfString ACCESS pMem + lSize;

			_pUtfString[0] := 16#0009;	// TAB

			lSize := lSize + 2;

		ELSE

			status := 2;
			RETURN;

		END_IF

		// Programmno

		brsitoa(CPRow.wProgramNo, ADR(_sValue));

		_lLen := LEN(_sValue);

		IF _lLen > 0 THEN

			IF (lSize + _lLen*2 ) <= lMaxSize THEN

				brwcsconv(pMem + lSize, ADR(_sValue), 0);

				lSize := lSize + 2* _lLen;

			ELSE

				status := 2;
				RETURN;

			END_IF

		END_IF

		IF (lSize + 2) <= lMaxSize THEN

			_pUtfString ACCESS pMem + lSize;

			_pUtfString[0] := 16#0009;	// TAB

			lSize := lSize + 2;

		ELSE

			status := 2;
			RETURN;

		END_IF

		// Zeitstempel

		_dttoa(dtTimestamp := CPRow.dtTimeStamp);

		IF (lSize + 38 ) <= lMaxSize THEN

			brwcsconv(pMem + lSize, ADR(_dttoa.sDateTime), 0);

			lSize := lSize + 38;

		ELSE

			status := 2;
			RETURN;

		END_IF

		IF (lSize + 2) <= lMaxSize THEN

			_pUtfString ACCESS pMem + lSize;

			_pUtfString[0] := 16#0009;	// TAB

			lSize := lSize + 2;

		ELSE

			status := 2;
			RETURN;

		END_IF

		// Soilfactor

		_sValue := REAL_TO_STRING(CPRow.rSoilfactor);

		_lLen := LEN(_sValue);

		IF _lLen > 0 THEN

			IF (lSize + _lLen*2 ) <= lMaxSize THEN

				brwcsconv(pMem + lSize, ADR(_sValue), 0);

				lSize := lSize + 2* _lLen;

			ELSE

				status := 2;
				RETURN;

			END_IF

		END_IF

		IF (lSize + 2) <= lMaxSize THEN

			_pUtfString ACCESS pMem + lSize;

			_pUtfString[0] := 16#0009;	// TAB

			lSize := lSize + 2;

		ELSE

			status := 2;
			RETURN;

		END_IF

		// Loadrate

		_sValue := UINT_TO_STRING(CPRow.wLoadrate);

		_lLen := LEN(_sValue);

		IF _lLen > 0 THEN

			IF (lSize + _lLen*2 ) <= lMaxSize THEN

				brwcsconv(pMem + lSize, ADR(_sValue), 0);

				lSize := lSize + 2* _lLen;

			ELSE

				status := 2;
				RETURN;

			END_IF

		END_IF

		IF (lSize + 2) <= lMaxSize THEN

			_pUtfString ACCESS pMem + lSize;

			_pUtfString[0] := 16#0009;	// TAB

			lSize := lSize + 2;

		ELSE

			status := 2;
			RETURN;

		END_IF

		// Foreground color

		_sValue := UINT_TO_STRING(CPRow.wColFor);

		_lLen := LEN(_sValue);

		IF _lLen > 0 THEN

			IF (lSize + _lLen*2 ) <= lMaxSize THEN

				brwcsconv(pMem + lSize, ADR(_sValue), 0);

				lSize := lSize + 2* _lLen;

			ELSE

				status := 2;
				RETURN;

			END_IF

		END_IF

		IF (lSize + 2) <= lMaxSize THEN

			_pUtfString ACCESS pMem + lSize;

			_pUtfString[0] := 16#0009;	// TAB

			lSize := lSize + 2;

		ELSE

			status := 2;
			RETURN;

		END_IF

		// Background color

		_sValue := UINT_TO_STRING(CPRow.wColBack);

		_lLen := LEN(_sValue);

		IF _lLen > 0 THEN

			IF (lSize + _lLen*2 ) <= lMaxSize THEN

				brwcsconv(pMem + lSize, ADR(_sValue), 0);

				lSize := lSize + 2* _lLen;

			ELSE

				status := 2;
				RETURN;

			END_IF

		END_IF

		IF (lSize + 4) <= lMaxSize THEN

			_pUtfString ACCESS pMem + lSize;

			_pUtfString[0] := 16#000D;	// Return
			_pUtfString[1] := 16#000A;	// Linefeed

			lSize := lSize + 4;

		ELSE

			status := 2;
			RETURN;

		END_IF

	ELSE

		status := ERR_FUB_ENABLE_FALSE;

	END_IF

END_FUNCTION_BLOCK
```

#### mnParam_WriteCSV80_Mem.st - String Daten schreiben
```iecst
(********************************************************************
 * COPYRIGHT -- Microsoft
 ********************************************************************
 * Library: mnParamLib
 * File: mnParam_WriteCSV80_Mem.st
 * Author: hunholz
 * Created: October 20, 2011
 ********************************************************************
 * Implementation of library mnParamLib
 ********************************************************************)

(* String Daten schreiben *)
FUNCTION_BLOCK mnParam_WriteCSV80_Mem

	IF enable THEN

		status := ERR_OK;

		IF pMem = 0 THEN

			status := 1;
			RETURN;

		END_IF

		IF (lSize + 6) <= lMaxSize THEN

			_pUtfString ACCESS pMem + lSize;

			_pUtfString[0] := 16#0038;	// 8
			_pUtfString[1] := 16#0030;	// 0
			_pUtfString[2] := 16#0009;	// TAB

			lSize := lSize + 6;

		ELSE

			status := 2;
			RETURN;

		END_IF

		// Container-ID

		brsitoa(ContentRow.iContainerID, ADR(_sValue));

		_lLen := LEN(_sValue);

		IF _lLen > 0 THEN

			IF (lSize + _lLen*2 ) <= lMaxSize THEN

				brwcsconv(pMem + lSize, ADR(_sValue), 0);

				lSize := lSize + 2* _lLen;

			ELSE

				status := 2;
				RETURN;

			END_IF

		END_IF

		IF (lSize + 2) <= lMaxSize THEN

			_pUtfString ACCESS pMem + lSize;

			_pUtfString[0] := 16#0009;	// TAB

			lSize := lSize + 2;

		ELSE

			status := 2;
			RETURN;

		END_IF

		// Instanz

		brsitoa(ContentRow.wInstance, ADR(_sValue));

		_lLen := LEN(_sValue);

		IF _lLen > 0 THEN

			IF (lSize + _lLen*2 ) <= lMaxSize THEN

				brwcsconv(pMem + lSize, ADR(_sValue), 0);

				lSize := lSize + 2* _lLen;

			ELSE

				status := 2;
				RETURN;

			END_IF

		END_IF

		IF (lSize + 2) <= lMaxSize THEN

			_pUtfString ACCESS pMem + lSize;

			_pUtfString[0] := 16#0009;	// TAB

			lSize := lSize + 2;

		ELSE

			status := 2;
			RETURN;

		END_IF

		// Zeitstempel

		_dttoa(dtTimestamp := ContentRow.dtTimestamp);

		IF (lSize + 38 ) <= lMaxSize THEN

			brwcsconv(pMem + lSize, ADR(_dttoa.sDateTime), 0);

			lSize := lSize + 38;

		ELSE

			status := 2;
			RETURN;

		END_IF

		IF (lSize + 4) <= lMaxSize THEN

			_pUtfString ACCESS pMem + lSize;

			_pUtfString[0] := 16#000D;	// Return
			_pUtfString[1] := 16#000A;	// Linefeed

			lSize := lSize + 4;

		ELSE

			status := 2;
			RETURN;

		END_IF

	ELSE

		status := ERR_FUB_ENABLE_FALSE;

	END_IF

END_FUNCTION_BLOCK
```

#### mnParam_WriteCSV90_Mem.st - String Daten schreiben
```iecst
(********************************************************************
 * COPYRIGHT -- Microsoft
 ********************************************************************
 * Library: mnParamLib
 * File: mnParam_WriteCSV90_Mem.st
 * Author: hunholz
 * Created: August 02, 2011
 ********************************************************************
 * Implementation of library mnParamLib
 ********************************************************************)

(* String Daten schreiben *)
FUNCTION_BLOCK mnParam_WriteCSV90_Mem

	IF enable THEN

		IF pMem = 0 THEN

			status := 1;
			RETURN;

		END_IF

		IF (lSize + 6) <= lMaxSize THEN

			_pUtfString ACCESS pMem + lSize;

			_pUtfString[0] := 16#0039;	// 9
			_pUtfString[1] := 16#0030;	// 0
			_pUtfString[2] := 16#0009;	// TAB

			lSize := lSize + 6;

		ELSE

			status := 2;
			RETURN;

		END_IF

		// IP-Adresse

		_lLen := brwcslen(ADR(IPRow.utfIP_Adress));

		IF _lLen > 0 THEN

			IF (lSize + _lLen*2 ) <= lMaxSize THEN

				brwcscpy(pMem + lSize, ADR(IPRow.utfIP_Adress));

				lSize := lSize + 2* _lLen;

			ELSE

				status := 2;
				RETURN;

			END_IF

		END_IF

		IF (lSize + 2) <= lMaxSize THEN

			_pUtfString ACCESS pMem + lSize;

			_pUtfString[0] := 16#0009;	// TAB

			lSize := lSize + 2;

		ELSE

			status := 2;
			RETURN;

		END_IF

		// Gateway

		_lLen := brwcslen(ADR(IPRow.utfGateway));

		IF _lLen > 0 THEN

			IF (lSize + _lLen*2 ) <= lMaxSize THEN

				brwcscpy(pMem + lSize, ADR(IPRow.utfGateway));

				lSize := lSize + 2* _lLen;

			ELSE

				status := 2;
				RETURN;

			END_IF

		END_IF

		IF (lSize + 4) <= lMaxSize THEN

			_pUtfString ACCESS pMem + lSize;

			_pUtfString[0] := 16#000D;	// Return
			_pUtfString[1] := 16#000A;	// Linefeed

			lSize := lSize + 4;

		ELSE

			status := 2;
			RETURN;

		END_IF

		status := 0;

	ELSE

		status := 65334;

	END_IF

END_FUNCTION_BLOCK
```

#### mnParam_WriteCSV251_Mem.st - Dateizeitstempel schreiben
```iecst
(********************************************************************
 * COPYRIGHT -- Microsoft
 ********************************************************************
 * Library: mnParamLib
 * File: mnParam_WriteCSV251_Mem.st
 * Author: hunholz
 * Created: August 02, 2011
 ********************************************************************
 * Implementation of library mnParamLib
 ********************************************************************)

(* Dateizeitstempel schreiben *)
FUNCTION_BLOCK mnParam_WriteCSV251_Mem

	IF enable THEN

		IF pMem = 0 THEN

			status := 1;
			RETURN;

		END_IF

		IF (lSize + 8) <= lMaxSize THEN

			_pUtfString ACCESS pMem + lSize;

			_pUtfString[0] := 16#0032;	// 2
			_pUtfString[1] := 16#0035;	// 5
			_pUtfString[2] := 16#0031;	// 1
			_pUtfString[3] := 16#0009;	// TAB

			lSize := lSize + 8;

		ELSE

			status := 2;
			RETURN;

		END_IF

		// Zeitstempel schreiben

		_dttoa(dtTimestamp := TimeRow.dtTimestamp);

		IF (lSize + 38 ) <= lMaxSize THEN

			brwcsconv(pMem + lSize, ADR(_dttoa.sDateTime), 0);

			lSize := lSize + 38;

		ELSE

			status := 2;
			RETURN;

		END_IF

		IF (lSize + 4) <= lMaxSize THEN

			_pUtfString ACCESS pMem + lSize;

			_pUtfString[0] := 16#000D;	// Return
			_pUtfString[1] := 16#000A;	// Linefeed

			lSize := lSize + 4;

		ELSE

			status := 2;
			RETURN;

		END_IF

		status := 0;

	ELSE

		status := 65334;

	END_IF

END_FUNCTION_BLOCK
```

#### mnParam_WriteCSV252_Mem.st - Zeile mit Maschinennummer
```iecst
(********************************************************************
 * COPYRIGHT -- Microsoft
 ********************************************************************
 * Library: mnParamLib
 * File: mnParam_WriteCSV252_Mem.st
 * Author: hunholz
 * Created: August 02, 2011
 ********************************************************************
 * Implementation of library mnParamLib
 ********************************************************************)

(* TODO: Add your comment here *)
FUNCTION_BLOCK mnParam_WriteCSV252_Mem

	IF enable THEN

		IF pMem = 0 THEN

			status := 1;
			RETURN;

		END_IF

		IF (lSize + 8) <= lMaxSize THEN

			_pUtfString ACCESS pMem + lSize;

			_pUtfString[0] := 16#0032;	// 2
			_pUtfString[1] := 16#0035;	// 5
			_pUtfString[2] := 16#0032;	// 2
			_pUtfString[3] := 16#0009;	// TAB

			lSize := lSize + 8;

		ELSE

			status := 2;
			RETURN;

		END_IF

		// Maschinennummer schreiben

		_lLen := brwcslen(ADR(MachineNoRow.utfMachineNo));

		IF _lLen > 0 THEN

			IF (lSize + _lLen*2 ) <= lMaxSize THEN

				brwcscpy(pMem + lSize, ADR(MachineNoRow.utfMachineNo));

				lSize := lSize + 2* _lLen;

			ELSE

				status := 2;
				RETURN;

			END_IF

		END_IF

		IF (lSize + 4) <= lMaxSize THEN

			_pUtfString ACCESS pMem + lSize;

			_pUtfString[0] := 16#000D;	// Return
			_pUtfString[1] := 16#000A;	// Linefeed

			lSize := lSize + 4;

		ELSE

			status := 2;
			RETURN;

		END_IF

		status := 0;

	ELSE

		status := 65334;

	END_IF

END_FUNCTION_BLOCK
```

#### mnParam_WriteCSV253_Mem.st - Versions Kopfzeile
```iecst
(********************************************************************
 * COPYRIGHT -- Microsoft
 ********************************************************************
 * Library: mnParamLib
 * File: mnParam_WriteCSV253_Mem.st
 * Author: hunholz
 * Created: August 02, 2011
 ********************************************************************
 * Implementation of library mnParamLib
 ********************************************************************)

(* Versions Kopfzeile *)
FUNCTION_BLOCK mnParam_WriteCSV253_Mem

	IF enable THEN

		IF pMem = 0 THEN

			status := 1;
			RETURN;

		END_IF

		IF (lSize + 8) <= lMaxSize THEN

			_pUtfString ACCESS pMem + lSize;

			_pUtfString[0] := 16#0032;	// 2
			_pUtfString[1] := 16#0035;	// 5
			_pUtfString[2] := 16#0033;	// 3
			_pUtfString[3] := 16#0009;	// TAB

			lSize := lSize + 8;

		ELSE

			status := 2;
			RETURN;

		END_IF

		// Version schreiben

		brsitoa(VersionRow.wVersion, ADR(_sVersion));

		IF LEN(_sVersion) > 0 THEN

			IF (lSize + LEN(_sVersion)*2 ) <= lMaxSize THEN

				brwcsconv(pMem + lSize, ADR(_sVersion), 0);

				lSize := lSize + 2*LEN(_sVersion);

			ELSE

				status := 2;
				RETURN;

			END_IF

		END_IF

		IF (lSize + 2) <= lMaxSize THEN

			_pUtfString ACCESS pMem + lSize;

			_pUtfString[0] := 16#0009;	// TAB

			lSize := lSize + 2;

		ELSE

			status := 2;
			RETURN;

		END_IF

		// Zeitstempel schreiben

		_dttoa(dtTimestamp := VersionRow.dtTimestamp);

		IF (lSize + 38 ) <= lMaxSize THEN

			brwcsconv(pMem + lSize, ADR(_dttoa.sDateTime), 0);

			lSize := lSize + 38;

		ELSE

			status := 2;
			RETURN;

		END_IF

		IF (lSize + 2) <= lMaxSize THEN

			_pUtfString ACCESS pMem + lSize;

			_pUtfString[0] := 16#0009;	// TAB

			lSize := lSize + 2;

		ELSE

			status := 2;
			RETURN;

		END_IF

		// Maschinentyp schreiben

		_lLen := brwcslen(ADR(VersionRow.utfMachineType));

		IF _lLen > 0 THEN

			IF (lSize + _lLen*2 ) <= lMaxSize THEN

				brwcscpy(pMem + lSize, ADR(VersionRow.utfMachineType));

				lSize := lSize + 2* _lLen;

			ELSE

				status := 2;
				RETURN;

			END_IF

		END_IF

		IF (lSize + 2) <= lMaxSize THEN

			_pUtfString ACCESS pMem + lSize;

			_pUtfString[0] := 16#0009;	// TAB

			lSize := lSize + 2;

		ELSE

			status := 2;
			RETURN;

		END_IF

		// Maschinensubtyp schreiben

		_lLen := brwcslen(ADR(VersionRow.utfMachineSubType));

		IF _lLen > 0 THEN

			IF (lSize + _lLen*2 ) <= lMaxSize THEN

				brwcscpy(pMem + lSize, ADR(VersionRow.utfMachineSubType));

				lSize := lSize + 2* _lLen;

			ELSE

				status := 2;
				RETURN;

			END_IF

		END_IF

		IF (lSize + 4) <= lMaxSize THEN

			_pUtfString ACCESS pMem + lSize;

			_pUtfString[0] := 16#000D;	// Return
			_pUtfString[1] := 16#000A;	// Linefeed

			lSize := lSize + 4;

		ELSE

			status := 2;
			RETURN;

		END_IF

		status := 0;

	ELSE

		status := 65334;

	END_IF

END_FUNCTION_BLOCK
```

#### mnParam_WriteCSV254_Mem.st - Kommentarzeile schreiben
```iecst
(********************************************************************
 * COPYRIGHT -- Microsoft
 ********************************************************************
 * Library: mnParamLib
 * File: mnParam_WriteCSV254_Mem.st
 * Author: hunholz
 * Created: August 01, 2011
 ********************************************************************
 * Implementation of library mnParamLib
 ********************************************************************)

(* Kommentarzeile schreiben *)
FUNCTION_BLOCK mnParam_WriteCSV254_Mem

	IF enable THEN

		IF pMem = 0 THEN

			status := 1;
			RETURN;

		END_IF

		IF (lSize + 8) <= lMaxSize THEN

			_pUtfString ACCESS pMem + lSize;

			_pUtfString[0] := 16#0032;	// 2
			_pUtfString[1] := 16#0035;	// 5
			_pUtfString[2] := 16#0034;	// 4
			_pUtfString[3] := 16#0009;	// TAB

			lSize := lSize + 8;

		ELSE

			status := 2;
			RETURN;

		END_IF

		IF LEN(sComment) > 0 THEN

			IF (lSize + LEN(sComment)*2 ) <= lMaxSize THEN

				brwcsconv(pMem + lSize, ADR(sComment), 0);

				lSize := lSize + 2*LEN(sComment);

			ELSE

				status := 2;
				RETURN;

			END_IF

		END_IF

		IF (lSize + 4) <= lMaxSize THEN

			_pUtfString ACCESS pMem + lSize;

			_pUtfString[0] := 16#000D;	// Return
			_pUtfString[1] := 16#000A;	// Linefeed

			lSize := lSize + 4;

		ELSE

			status := 2;
			RETURN;

		END_IF

		status := 0;

	ELSE

		status := 65334;

	END_IF

END_FUNCTION_BLOCK
```

#### mnParam_WriteCSV255_Mem.st - File-Ende schreiben
```iecst
(********************************************************************
 * COPYRIGHT -- Microsoft
 ********************************************************************
 * Library: mnParamLib
 * File: mnParam_WriteCSV255_Mem.st
 * Author: hunholz
 * Created: August 01, 2011
 ********************************************************************
 * Implementation of library mnParamLib
 ********************************************************************)

(* File-Ende schreiben *)
FUNCTION_BLOCK mnParam_WriteCSV255_Mem

	IF enable THEN

		IF pMem = 0 THEN

			status := 1;
			RETURN;

		END_IF

		IF (lSize + 10) > lMaxSize THEN

			_pUtfString ACCESS pMem + lSize;

			_pUtfString[0] := 16#0032;	// 2
			_pUtfString[1] := 16#0035;	// 5
			_pUtfString[2] := 16#0035;	// 5
			_pUtfString[3] := 16#000D;	// Return
			_pUtfString[4] := 16#000A;	// Linefeed

			lSize := lSize + 10;

		ELSE

			status := 2;
			RETURN;

		END_IF

		status := 0;

	ELSE

		status := 65334;

	END_IF

END_FUNCTION_BLOCK
```

#### mnParam_datetimetoa.st - Wandelt Datum Zeit in ISO String
```iecst
(********************************************************************
 * COPYRIGHT -- Microsoft
 ********************************************************************
 * Library: mnParamLib
 * File: mnParam_datetimetoa.st
 * Author: hunholz
 * Created: August 02, 2011
 ********************************************************************
 * Implementation of library mnParamLib
 ********************************************************************)

(* Wandelt Datum Zeit in ISO String *)
FUNCTION_BLOCK mnParam_datetimetoa

	brsmemset(ADR(_s2dig),0,SIZEOF(_s2dig));
	_b2dig ACCESS ADR(_s2dig);

	DT_TO_DTStructure(DT1 := dtTimestamp, ADR(_dtStruc));

	brsitoa(_dtStruc.year, ADR(sDateTime));

	brsstrcat(ADR(sDateTime), ADR('-'));

	_b2dig[0] := (_dtStruc.month / 10) + 16#30;
	_b2dig[1] := (_dtStruc.month MOD 10) + 16#30;

	brsstrcat(ADR(sDateTime), ADR(_s2dig));
	brsstrcat(ADR(sDateTime), ADR('-'));

	_b2dig[0] := (_dtStruc.day / 10) + 16#30;
	_b2dig[1] := (_dtStruc.day MOD 10) + 16#30;

	brsstrcat(ADR(sDateTime), ADR(_s2dig));
	brsstrcat(ADR(sDateTime), ADR('T'));

	_b2dig[0] := (_dtStruc.hour / 10) + 16#30;
	_b2dig[1] := (_dtStruc.hour MOD 10) + 16#30;

	brsstrcat(ADR(sDateTime), ADR(_s2dig));
	brsstrcat(ADR(sDateTime), ADR(':'));

	_b2dig[0] := (_dtStruc.minute / 10) + 16#30;
	_b2dig[1] := (_dtStruc.minute MOD 10) + 16#30;

	brsstrcat(ADR(sDateTime), ADR(_s2dig));
	brsstrcat(ADR(sDateTime), ADR(':'));

	_b2dig[0] := (_dtStruc.second / 10) + 16#30;
	_b2dig[1] := (_dtStruc.second MOD 10) + 16#30;

	brsstrcat(ADR(sDateTime), ADR(_s2dig));

END_FUNCTION_BLOCK
```

#### mnParam_datetoa.st - Wandelt Datum Zeit in ISO String
```iecst
(********************************************************************
 * COPYRIGHT -- Microsoft
 ********************************************************************
 * Library: mnParamLib
 * File: mnParam_datetoa.st
 * Author: hunholz
 * Created: Mar 23, 2012
 ********************************************************************
 * Implementation of library mnParamLib
 ********************************************************************)

(* Wandelt Datum in ISO String *)
FUNCTION_BLOCK mnParam_datetoa

	brsmemset(ADR(_s2dig),0,SIZEOF(_s2dig));
	_b2dig ACCESS ADR(_s2dig);

	DT_TO_DTStructure(DT1 := dtTimestamp, ADR(_dtStruc));

	brsitoa(_dtStruc.year, ADR(sDate));

	brsstrcat(ADR(sDate), ADR('-'));

	_b2dig[0] := (_dtStruc.month / 10) + 16#30;
	_b2dig[1] := (_dtStruc.month MOD 10) + 16#30;

	brsstrcat(ADR(sDate), ADR(_s2dig));
	brsstrcat(ADR(sDate), ADR('-'));

	_b2dig[0] := (_dtStruc.day / 10) + 16#30;
	_b2dig[1] := (_dtStruc.day MOD 10) + 16#30;

	brsstrcat(ADR(sDate), ADR(_s2dig));

END_FUNCTION_BLOCK
```
